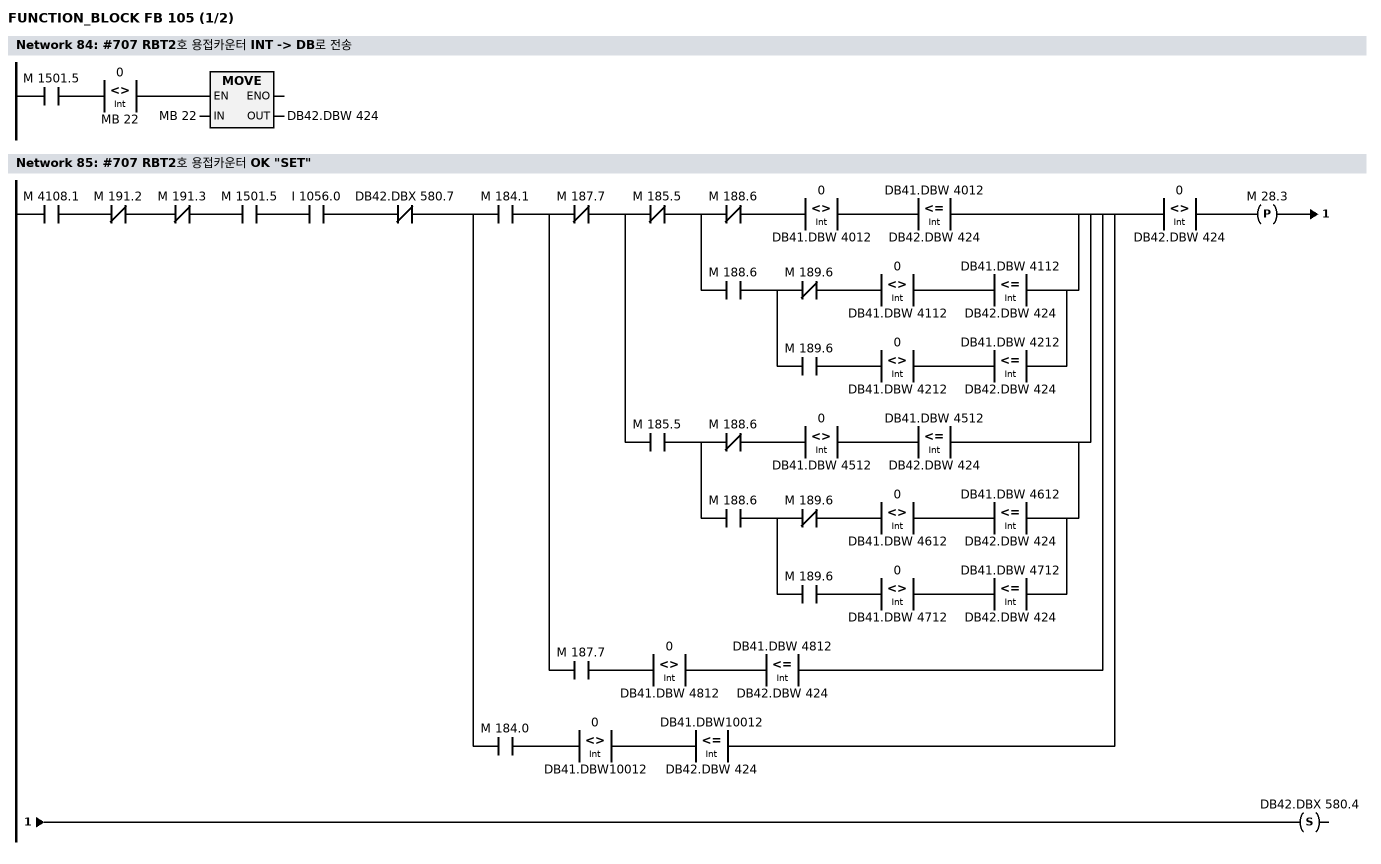

      A     M   1501.5;
      A(    ;
      L     0;
      L     MB    22;
      <>I   ;
      )     ;
      JNB   _093;
      L     MB    22;
      T     DB42.DBW  424;
_093: NOP   0;
NETWORK
TITLE =#707 RBT2호 용접카운터 OK "SET"

      A     M   4108.1;
      AN    M    191.2;
      AN    M    191.3;
      A     M   1501.5;
      A     I   1056.0;
      AN    DB42.DBX  580.7;
      A(    ;
      A     M    184.1;
      A(    ;
      AN    M    187.7;
      A(    ;
      AN    M    185.5;
      A(    ;
      AN    M    188.6;
      A(    ;
      L     0;
      L     DB41.DBW 4012;
      <>I   ;
      )     ;
      A(    ;
      L     DB41.DBW 4012;
      L     DB42.DBW  424;
      <=I   ;
      )     ;
      O     ;
      A     M    188.6;
      A(    ;
      AN    M    189.6;
      A(    ;
      L     0;
      L     DB41.DBW 4112;
      <>I   ;
      )     ;
      A(    ;
      L     DB41.DBW 4112;
      L     DB42.DBW  424;
      <=I   ;
      )     ;
      O     ;
      A     M    189.6;
      A(    ;
      L     0;
      L     DB41.DBW 4212;
      <>I   ;
      )     ;
      A(    ;
      L     DB41.DBW 4212;
      L     DB42.DBW  424;
      <=I   ;
      )     ;
      )     ;
      )     ;
      O     ;
      A     M    185.5;
      A(    ;
      AN    M    188.6;
      A(    ;
      L     0;
      L     DB41.DBW 4512;
      <>I   ;
      )     ;
      A(    ;
      L     DB41.DBW 4512;
      L     DB42.DBW  424;
      <=I   ;
      )     ;
      O     ;
      A     M    188.6;
      A(    ;
      AN    M    189.6;
      A(    ;
      L     0;
      L     DB41.DBW 4612;
      <>I   ;
      )     ;
      A(    ;
      L     DB41.DBW 4612;
      L     DB42.DBW  424;
      <=I   ;
      )     ;
      O     ;
      A     M    189.6;
      A(    ;
      L     0;
      L     DB41.DBW 4712;
      <>I   ;
      )     ;
      A(    ;
      L     DB41.DBW 4712;
      L     DB42.DBW  424;
      <=I   ;
      )     ;
      )     ;
      )     ;
      )     ;
      O     ;
      A     M    187.7;
      A(    ;
      L     0;
      L     DB41.DBW 4812;
      <>I   ;
      )     ;
      A(    ;
      L     DB41.DBW 4812;
      L     DB42.DBW  424;
      <=I   ;
      )     ;
      )     ;
      O     ;
      A     M    184.0;
      A(    ;
      L     0;
      L     DB41.DBW10012;
      <>I   ;
      )     ;
      A(    ;
      L     DB41.DBW10012;
      L     DB42.DBW  424;
      <=I   ;
      )     ;
      )     ;
      A(    ;
      L     0;
      L     DB42.DBW  424;
      <>I   ;
      )     ;
      FP    M     28.3;
      S     DB42.DBX  580.4;
NETWORK
TITLE =#707 RBT2호 용접카운터 NG "SET"
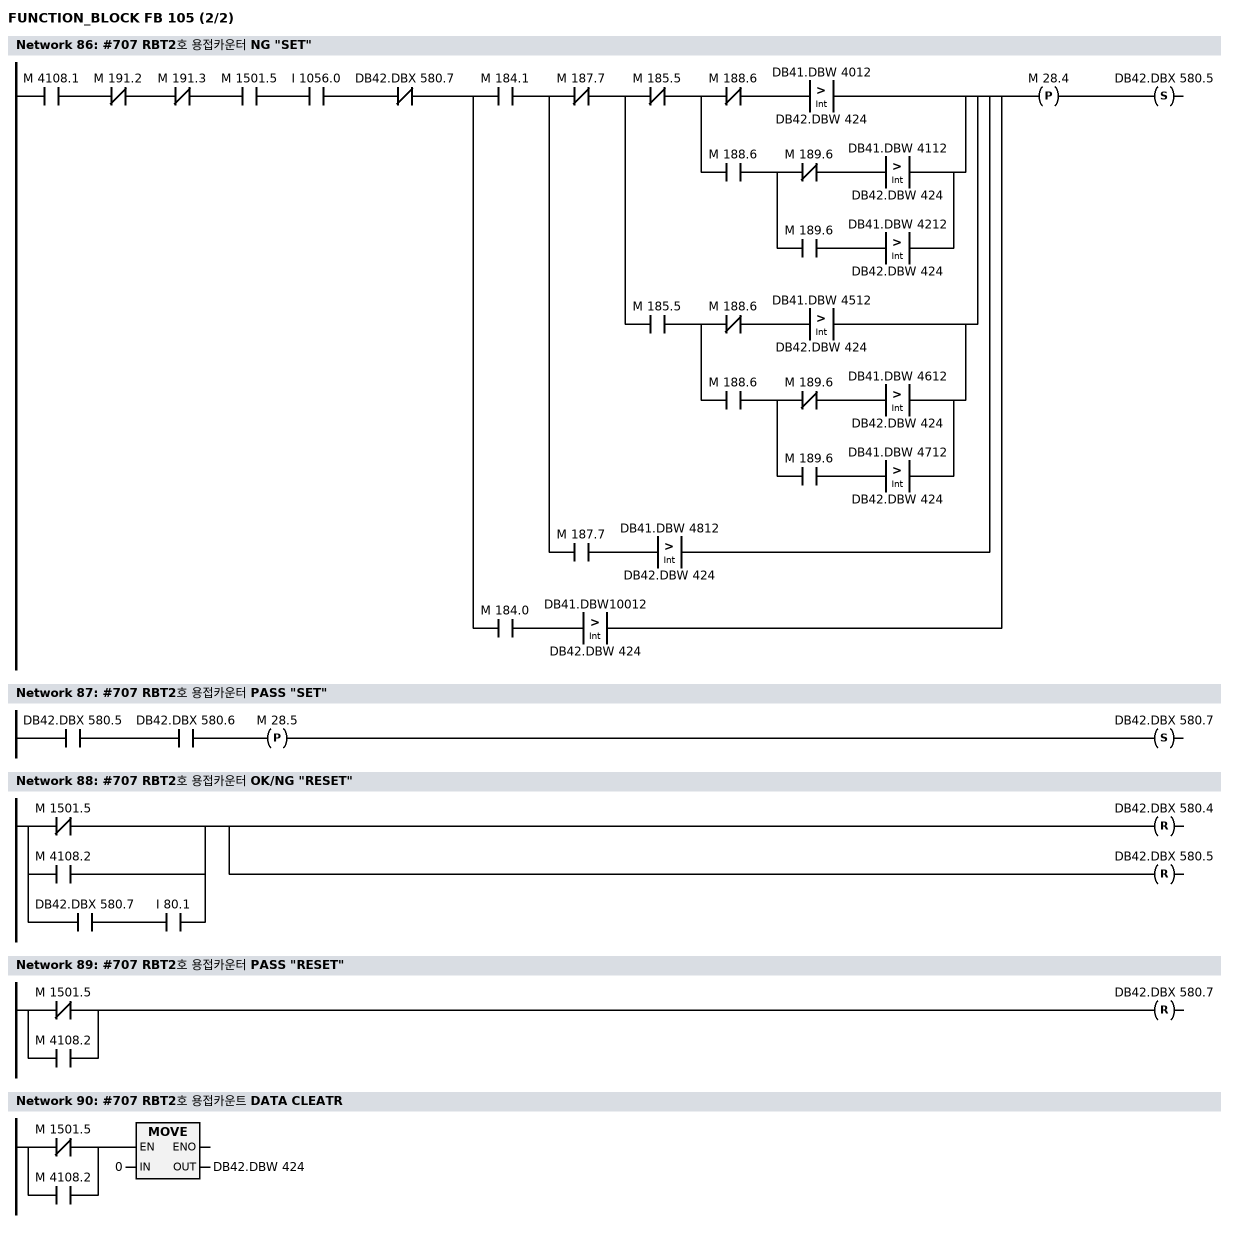

      A     M   4108.1;
      AN    M    191.2;
      AN    M    191.3;
      A     M   1501.5;
      A     I   1056.0;
      AN    DB42.DBX  580.7;
      A(    ;
      A     M    184.1;
      A(    ;
      AN    M    187.7;
      A(    ;
      AN    M    185.5;
      A(    ;
      AN    M    188.6;
      A(    ;
      L     DB41.DBW 4012;
      L     DB42.DBW  424;
      >I    ;
      )     ;
      O     ;
      A     M    188.6;
      A(    ;
      AN    M    189.6;
      A(    ;
      L     DB41.DBW 4112;
      L     DB42.DBW  424;
      >I    ;
      )     ;
      O     ;
      A     M    189.6;
      A(    ;
      L     DB41.DBW 4212;
      L     DB42.DBW  424;
      >I    ;
      )     ;
      )     ;
      )     ;
      O     ;
      A     M    185.5;
      A(    ;
      AN    M    188.6;
      A(    ;
      L     DB41.DBW 4512;
      L     DB42.DBW  424;
      >I    ;
      )     ;
      O     ;
      A     M    188.6;
      A(    ;
      AN    M    189.6;
      A(    ;
      L     DB41.DBW 4612;
      L     DB42.DBW  424;
      >I    ;
      )     ;
      O     ;
      A     M    189.6;
      A(    ;
      L     DB41.DBW 4712;
      L     DB42.DBW  424;
      >I    ;
      )     ;
      )     ;
      )     ;
      )     ;
      O     ;
      A     M    187.7;
      A(    ;
      L     DB41.DBW 4812;
      L     DB42.DBW  424;
      >I    ;
      )     ;
      )     ;
      O     ;
      A     M    184.0;
      A(    ;
      L     DB41.DBW10012;
      L     DB42.DBW  424;
      >I    ;
      )     ;
      )     ;
      FP    M     28.4;
      S     DB42.DBX  580.5;
NETWORK
TITLE =#707 RBT2호 용접카운터 PASS "SET"
//
//
      A     DB42.DBX  580.5;
      A     DB42.DBX  580.6;
      FP    M     28.5;
      S     DB42.DBX  580.7;
NETWORK
TITLE =#707 RBT2호 용접카운터 OK/NG "RESET"

      ON    M   1501.5;
      O     M   4108.2;
      O     ;
      A     DB42.DBX  580.7;
      A     I     80.1;
      R     DB42.DBX  580.4;
      R     DB42.DBX  580.5;
NETWORK
TITLE =#707 RBT2호 용접카운터 PASS "RESET"

      ON    M   1501.5;
      O     M   4108.2;
      R     DB42.DBX  580.7;
NETWORK
TITLE =#707 RBT2호 용접카운트 DATA CLEATR

      A(    ;
      ON    M   1501.5;
      O     M   4108.2;
      )     ;
      JNB   _094;
      L     0;
      T     DB42.DBW  424;
_094: NOP   0;
NETWORK
TITLE =#707 RBT3호 용접카운터 INT -> DB로 전송보조

      AN    OV;
      =     L      2.0;
      A     L      2.0;
      A     I   1068.0;
      =     M     23.0;
      A     L      2.0;
      A     I   1068.1;
      =     M     23.1;
      A     L      2.0;
      A     I   1068.2;
      =     M     23.2;
      A     L      2.0;
      A     I   1068.3;
      =     M     23.3;
      A     L      2.0;
      A     I   1068.4;
      =     M     23.4;
      A     L      2.0;
      AN    M      3.3;
      =     L      2.1;
      A     L      2.1;
      A     I   1068.5;
      =     M     23.5;
      A     L      2.1;
      A     I   1068.6;
      =     M     23.6;
      A     L      2.1;
      A     I   1068.7;
      =     M     23.7;
NETWORK
TITLE =#707 RBT3호 용접카운터 INT -> DB로 전송
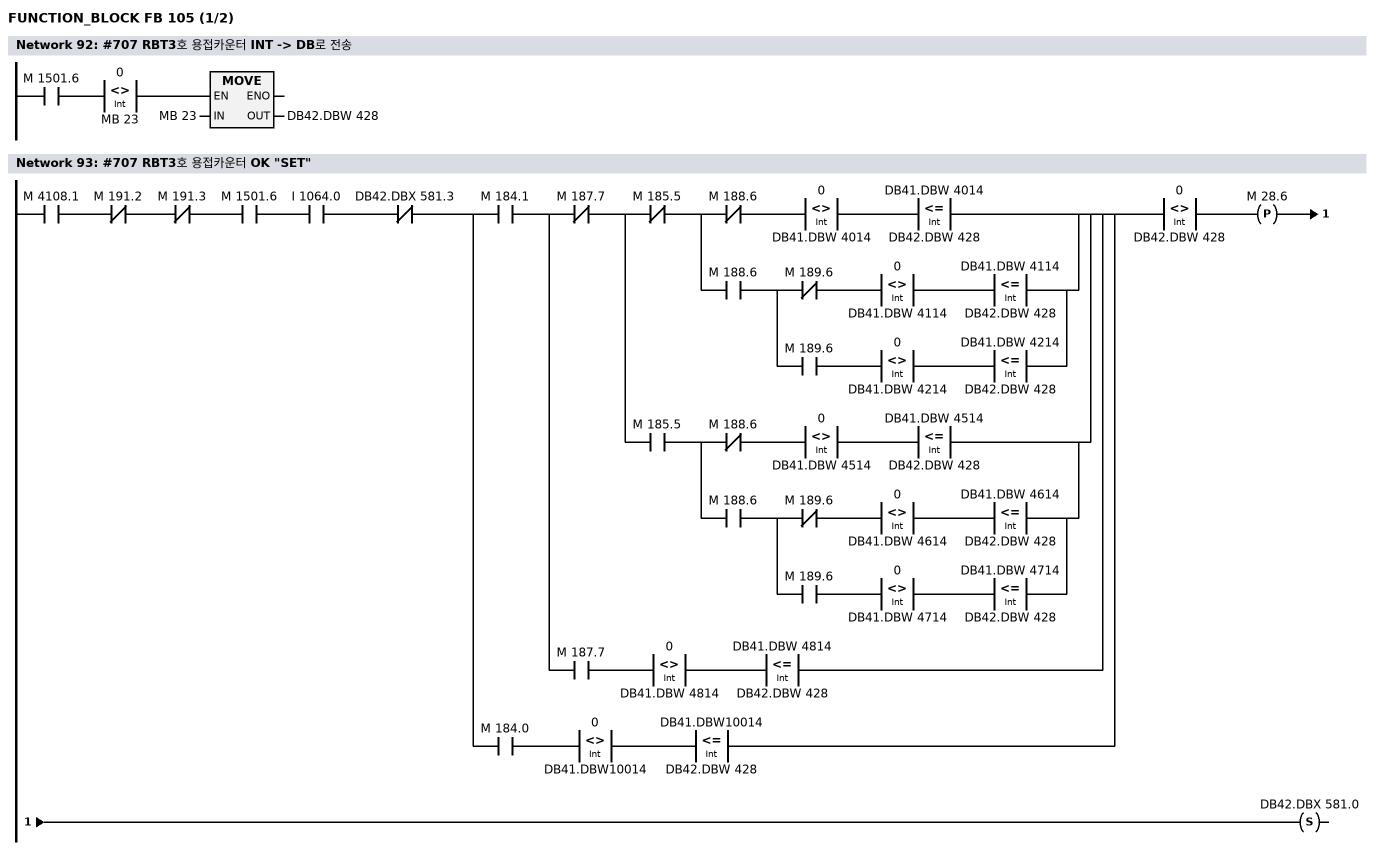

      A     M   1501.6;
      A(    ;
      L     0;
      L     MB    23;
      <>I   ;
      )     ;
      JNB   _095;
      L     MB    23;
      T     DB42.DBW  428;
_095: NOP   0;
NETWORK
TITLE =#707 RBT3호 용접카운터 OK "SET"

      A     M   4108.1;
      AN    M    191.2;
      AN    M    191.3;
      A     M   1501.6;
      A     I   1064.0;
      AN    DB42.DBX  581.3;
      A(    ;
      A     M    184.1;
      A(    ;
      AN    M    187.7;
      A(    ;
      AN    M    185.5;
      A(    ;
      AN    M    188.6;
      A(    ;
      L     0;
      L     DB41.DBW 4014;
      <>I   ;
      )     ;
      A(    ;
      L     DB41.DBW 4014;
      L     DB42.DBW  428;
      <=I   ;
      )     ;
      O     ;
      A     M    188.6;
      A(    ;
      AN    M    189.6;
      A(    ;
      L     0;
      L     DB41.DBW 4114;
      <>I   ;
      )     ;
      A(    ;
      L     DB41.DBW 4114;
      L     DB42.DBW  428;
      <=I   ;
      )     ;
      O     ;
      A     M    189.6;
      A(    ;
      L     0;
      L     DB41.DBW 4214;
      <>I   ;
      )     ;
      A(    ;
      L     DB41.DBW 4214;
      L     DB42.DBW  428;
      <=I   ;
      )     ;
      )     ;
      )     ;
      O     ;
      A     M    185.5;
      A(    ;
      AN    M    188.6;
      A(    ;
      L     0;
      L     DB41.DBW 4514;
      <>I   ;
      )     ;
      A(    ;
      L     DB41.DBW 4514;
      L     DB42.DBW  428;
      <=I   ;
      )     ;
      O     ;
      A     M    188.6;
      A(    ;
      AN    M    189.6;
      A(    ;
      L     0;
      L     DB41.DBW 4614;
      <>I   ;
      )     ;
      A(    ;
      L     DB41.DBW 4614;
      L     DB42.DBW  428;
      <=I   ;
      )     ;
      O     ;
      A     M    189.6;
      A(    ;
      L     0;
      L     DB41.DBW 4714;
      <>I   ;
      )     ;
      A(    ;
      L     DB41.DBW 4714;
      L     DB42.DBW  428;
      <=I   ;
      )     ;
      )     ;
      )     ;
      )     ;
      O     ;
      A     M    187.7;
      A(    ;
      L     0;
      L     DB41.DBW 4814;
      <>I   ;
      )     ;
      A(    ;
      L     DB41.DBW 4814;
      L     DB42.DBW  428;
      <=I   ;
      )     ;
      )     ;
      O     ;
      A     M    184.0;
      A(    ;
      L     0;
      L     DB41.DBW10014;
      <>I   ;
      )     ;
      A(    ;
      L     DB41.DBW10014;
      L     DB42.DBW  428;
      <=I   ;
      )     ;
      )     ;
      A(    ;
      L     0;
      L     DB42.DBW  428;
      <>I   ;
      )     ;
      FP    M     28.6;
      S     DB42.DBX  581.0;
NETWORK
TITLE =#707 RBT3호 용접카운터 NG "SET"
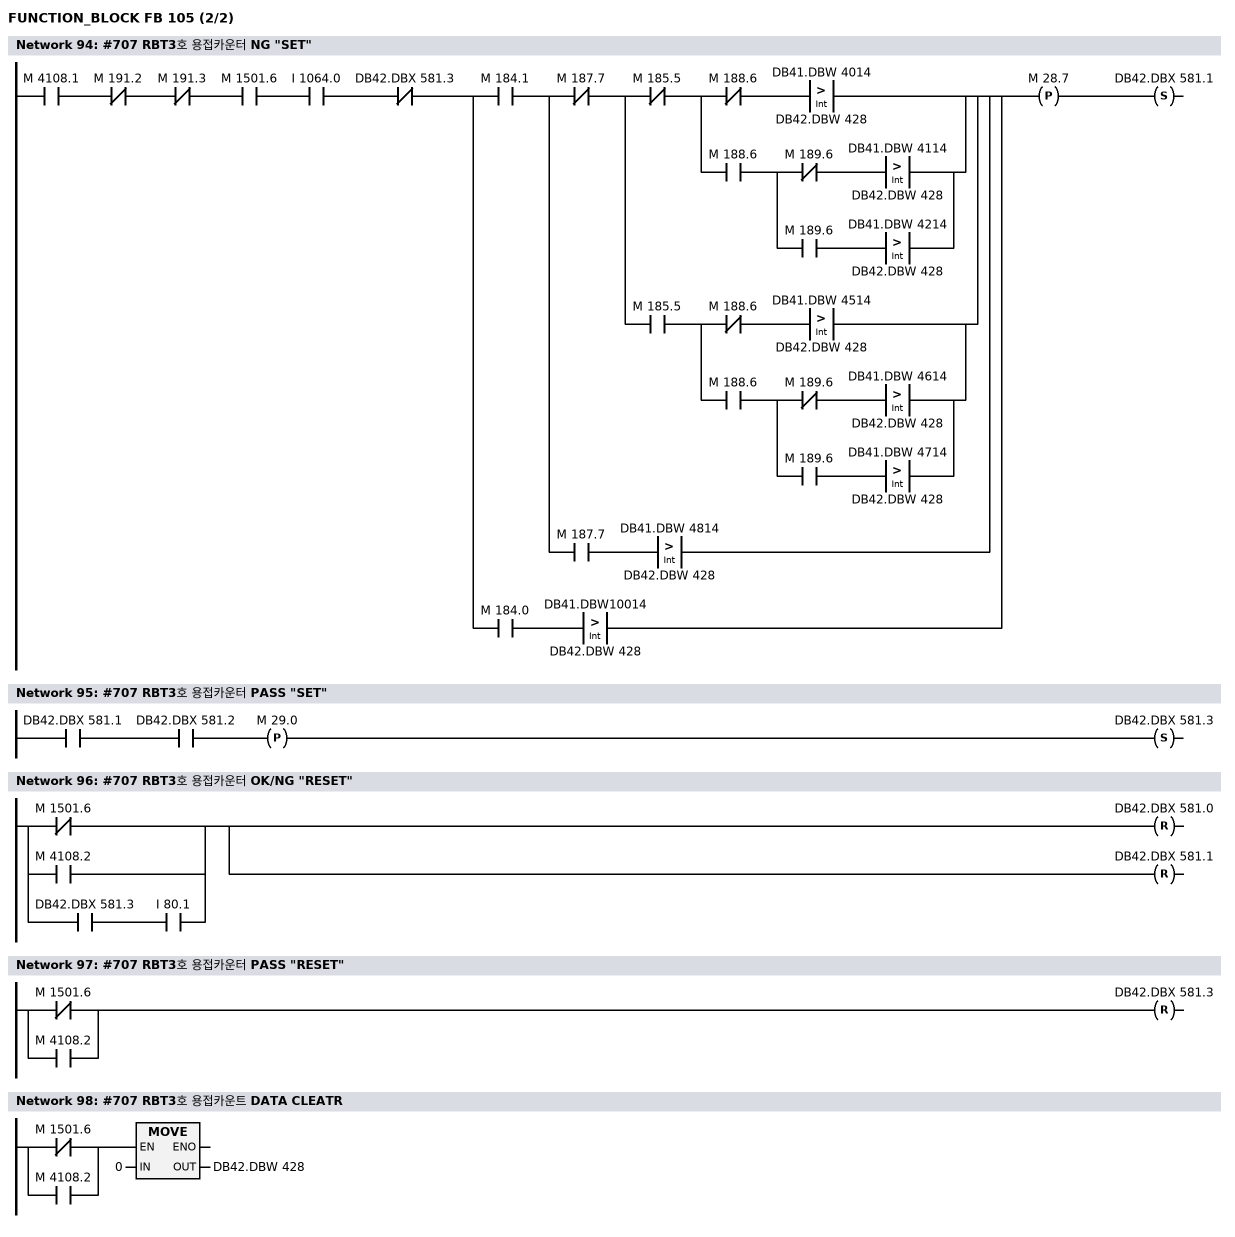

      A     M   4108.1;
      AN    M    191.2;
      AN    M    191.3;
      A     M   1501.6;
      A     I   1064.0;
      AN    DB42.DBX  581.3;
      A(    ;
      A     M    184.1;
      A(    ;
      AN    M    187.7;
      A(    ;
      AN    M    185.5;
      A(    ;
      AN    M    188.6;
      A(    ;
      L     DB41.DBW 4014;
      L     DB42.DBW  428;
      >I    ;
      )     ;
      O     ;
      A     M    188.6;
      A(    ;
      AN    M    189.6;
      A(    ;
      L     DB41.DBW 4114;
      L     DB42.DBW  428;
      >I    ;
      )     ;
      O     ;
      A     M    189.6;
      A(    ;
      L     DB41.DBW 4214;
      L     DB42.DBW  428;
      >I    ;
      )     ;
      )     ;
      )     ;
      O     ;
      A     M    185.5;
      A(    ;
      AN    M    188.6;
      A(    ;
      L     DB41.DBW 4514;
      L     DB42.DBW  428;
      >I    ;
      )     ;
      O     ;
      A     M    188.6;
      A(    ;
      AN    M    189.6;
      A(    ;
      L     DB41.DBW 4614;
      L     DB42.DBW  428;
      >I    ;
      )     ;
      O     ;
      A     M    189.6;
      A(    ;
      L     DB41.DBW 4714;
      L     DB42.DBW  428;
      >I    ;
      )     ;
      )     ;
      )     ;
      )     ;
      O     ;
      A     M    187.7;
      A(    ;
      L     DB41.DBW 4814;
      L     DB42.DBW  428;
      >I    ;
      )     ;
      )     ;
      O     ;
      A     M    184.0;
      A(    ;
      L     DB41.DBW10014;
      L     DB42.DBW  428;
      >I    ;
      )     ;
      )     ;
      FP    M     28.7;
      S     DB42.DBX  581.1;
NETWORK
TITLE =#707 RBT3호 용접카운터 PASS "SET"
//
//
      A     DB42.DBX  581.1;
      A     DB42.DBX  581.2;
      FP    M     29.0;
      S     DB42.DBX  581.3;
NETWORK
TITLE =#707 RBT3호 용접카운터 OK/NG "RESET"

      ON    M   1501.6;
      O     M   4108.2;
      O     ;
      A     DB42.DBX  581.3;
      A     I     80.1;
      R     DB42.DBX  581.0;
      R     DB42.DBX  581.1;
NETWORK
TITLE =#707 RBT3호 용접카운터 PASS "RESET"

      ON    M   1501.6;
      O     M   4108.2;
      R     DB42.DBX  581.3;
NETWORK
TITLE =#707 RBT3호 용접카운트 DATA CLEATR

      A(    ;
      ON    M   1501.6;
      O     M   4108.2;
      )     ;
      JNB   _096;
      L     0;
      T     DB42.DBW  428;
_096: NOP   0;
NETWORK
TITLE =#707 RBT4호 용접카운터 INT -> DB로 전송보조

      AN    OV;
      =     L      2.0;
      A     L      2.0;
      A     I   1076.0;
      =     M     24.0;
      A     L      2.0;
      A     I   1076.1;
      =     M     24.1;
      A     L      2.0;
      A     I   1076.2;
      =     M     24.2;
      A     L      2.0;
      A     I   1076.3;
      =     M     24.3;
      A     L      2.0;
      A     I   1076.4;
      =     M     24.4;
      A     L      2.0;
      AN    M      3.3;
      =     L      2.1;
      A     L      2.1;
      A     I   1076.5;
      =     M     24.5;
      A     L      2.1;
      A     I   1076.6;
      =     M     24.6;
      A     L      2.1;
      A     I   1076.7;
      =     M     24.7;
NETWORK
TITLE =#707 RBT4호 용접카운터 INT -> DB로 전송
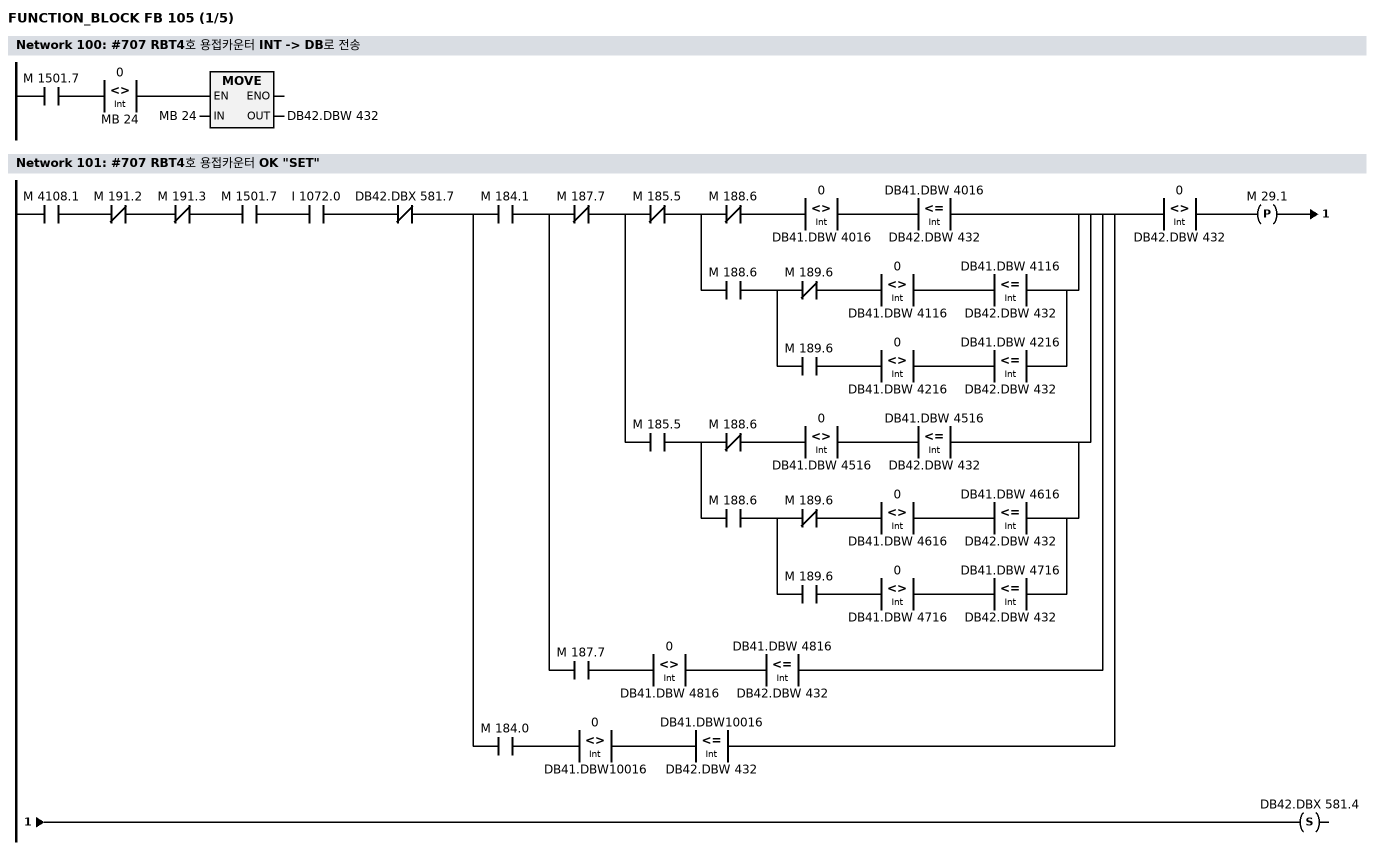

      A     M   1501.7;
      A(    ;
      L     0;
      L     MB    24;
      <>I   ;
      )     ;
      JNB   _097;
      L     MB    24;
      T     DB42.DBW  432;
_097: NOP   0;
NETWORK
TITLE =#707 RBT4호 용접카운터 OK "SET"

      A     M   4108.1;
      AN    M    191.2;
      AN    M    191.3;
      A     M   1501.7;
      A     I   1072.0;
      AN    DB42.DBX  581.7;
      A(    ;
      A     M    184.1;
      A(    ;
      AN    M    187.7;
      A(    ;
      AN    M    185.5;
      A(    ;
      AN    M    188.6;
      A(    ;
      L     0;
      L     DB41.DBW 4016;
      <>I   ;
      )     ;
      A(    ;
      L     DB41.DBW 4016;
      L     DB42.DBW  432;
      <=I   ;
      )     ;
      O     ;
      A     M    188.6;
      A(    ;
      AN    M    189.6;
      A(    ;
      L     0;
      L     DB41.DBW 4116;
      <>I   ;
      )     ;
      A(    ;
      L     DB41.DBW 4116;
      L     DB42.DBW  432;
      <=I   ;
      )     ;
      O     ;
      A     M    189.6;
      A(    ;
      L     0;
      L     DB41.DBW 4216;
      <>I   ;
      )     ;
      A(    ;
      L     DB41.DBW 4216;
      L     DB42.DBW  432;
      <=I   ;
      )     ;
      )     ;
      )     ;
      O     ;
      A     M    185.5;
      A(    ;
      AN    M    188.6;
      A(    ;
      L     0;
      L     DB41.DBW 4516;
      <>I   ;
      )     ;
      A(    ;
      L     DB41.DBW 4516;
      L     DB42.DBW  432;
      <=I   ;
      )     ;
      O     ;
      A     M    188.6;
      A(    ;
      AN    M    189.6;
      A(    ;
      L     0;
      L     DB41.DBW 4616;
      <>I   ;
      )     ;
      A(    ;
      L     DB41.DBW 4616;
      L     DB42.DBW  432;
      <=I   ;
      )     ;
      O     ;
      A     M    189.6;
      A(    ;
      L     0;
      L     DB41.DBW 4716;
      <>I   ;
      )     ;
      A(    ;
      L     DB41.DBW 4716;
      L     DB42.DBW  432;
      <=I   ;
      )     ;
      )     ;
      )     ;
      )     ;
      O     ;
      A     M    187.7;
      A(    ;
      L     0;
      L     DB41.DBW 4816;
      <>I   ;
      )     ;
      A(    ;
      L     DB41.DBW 4816;
      L     DB42.DBW  432;
      <=I   ;
      )     ;
      )     ;
      O     ;
      A     M    184.0;
      A(    ;
      L     0;
      L     DB41.DBW10016;
      <>I   ;
      )     ;
      A(    ;
      L     DB41.DBW10016;
      L     DB42.DBW  432;
      <=I   ;
      )     ;
      )     ;
      A(    ;
      L     0;
      L     DB42.DBW  432;
      <>I   ;
      )     ;
      FP    M     29.1;
      S     DB42.DBX  581.4;
NETWORK
TITLE =#707 RBT4호 용접카운터 NG "SET"
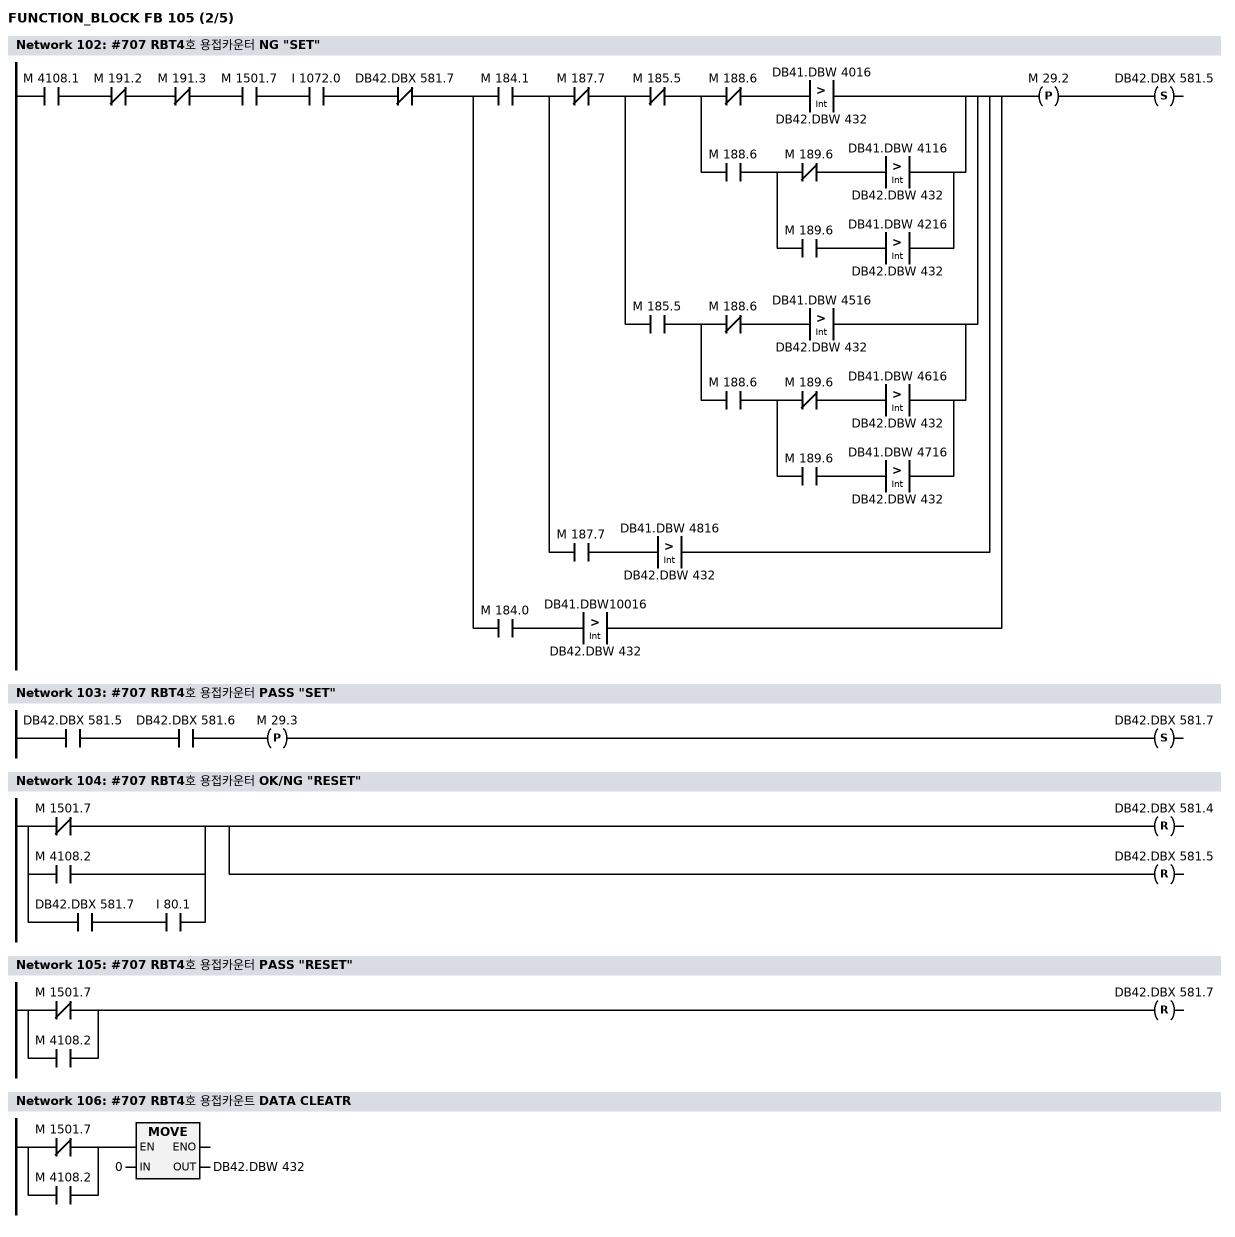

      A     M   4108.1;
      AN    M    191.2;
      AN    M    191.3;
      A     M   1501.7;
      A     I   1072.0;
      AN    DB42.DBX  581.7;
      A(    ;
      A     M    184.1;
      A(    ;
      AN    M    187.7;
      A(    ;
      AN    M    185.5;
      A(    ;
      AN    M    188.6;
      A(    ;
      L     DB41.DBW 4016;
      L     DB42.DBW  432;
      >I    ;
      )     ;
      O     ;
      A     M    188.6;
      A(    ;
      AN    M    189.6;
      A(    ;
      L     DB41.DBW 4116;
      L     DB42.DBW  432;
      >I    ;
      )     ;
      O     ;
      A     M    189.6;
      A(    ;
      L     DB41.DBW 4216;
      L     DB42.DBW  432;
      >I    ;
      )     ;
      )     ;
      )     ;
      O     ;
      A     M    185.5;
      A(    ;
      AN    M    188.6;
      A(    ;
      L     DB41.DBW 4516;
      L     DB42.DBW  432;
      >I    ;
      )     ;
      O     ;
      A     M    188.6;
      A(    ;
      AN    M    189.6;
      A(    ;
      L     DB41.DBW 4616;
      L     DB42.DBW  432;
      >I    ;
      )     ;
      O     ;
      A     M    189.6;
      A(    ;
      L     DB41.DBW 4716;
      L     DB42.DBW  432;
      >I    ;
      )     ;
      )     ;
      )     ;
      )     ;
      O     ;
      A     M    187.7;
      A(    ;
      L     DB41.DBW 4816;
      L     DB42.DBW  432;
      >I    ;
      )     ;
      )     ;
      O     ;
      A     M    184.0;
      A(    ;
      L     DB41.DBW10016;
      L     DB42.DBW  432;
      >I    ;
      )     ;
      )     ;
      FP    M     29.2;
      S     DB42.DBX  581.5;
NETWORK
TITLE =#707 RBT4호 용접카운터 PASS "SET"
//
//
      A     DB42.DBX  581.5;
      A     DB42.DBX  581.6;
      FP    M     29.3;
      S     DB42.DBX  581.7;
NETWORK
TITLE =#707 RBT4호 용접카운터 OK/NG "RESET"

      ON    M   1501.7;
      O     M   4108.2;
      O     ;
      A     DB42.DBX  581.7;
      A     I     80.1;
      R     DB42.DBX  581.4;
      R     DB42.DBX  581.5;
NETWORK
TITLE =#707 RBT4호 용접카운터 PASS "RESET"

      ON    M   1501.7;
      O     M   4108.2;
      R     DB42.DBX  581.7;
NETWORK
TITLE =#707 RBT4호 용접카운트 DATA CLEATR

      A(    ;
      ON    M   1501.7;
      O     M   4108.2;
      )     ;
      JNB   _098;
      L     0;
      T     DB42.DBW  432;
_098: NOP   0;
NETWORK
TITLE =
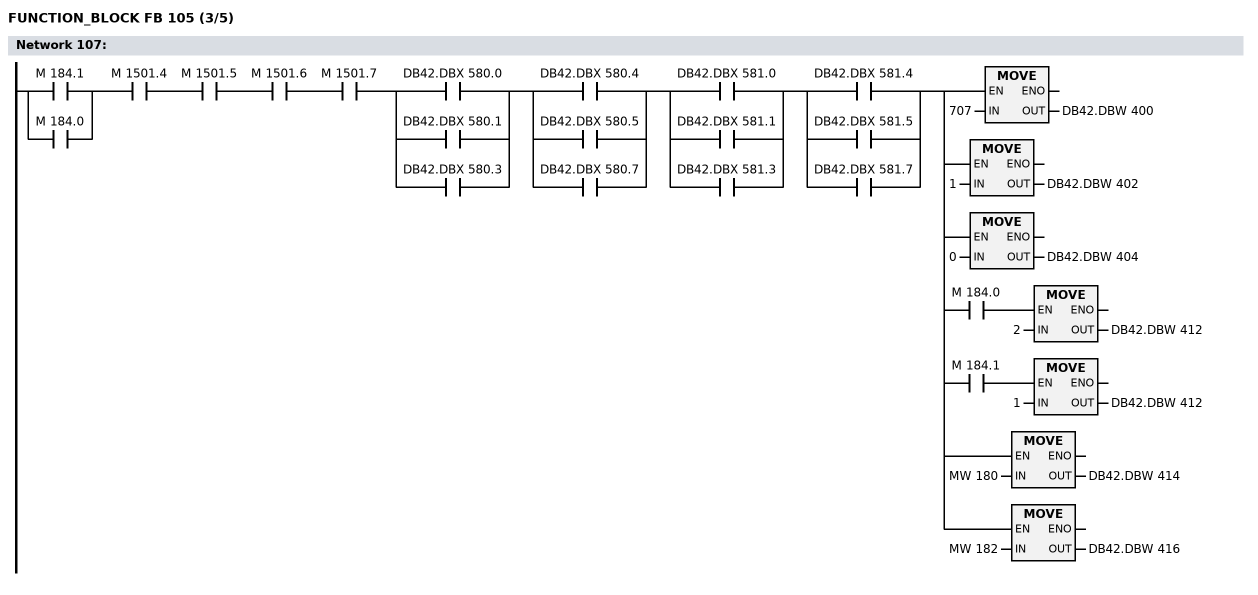

      A(    ;
      O     M    184.1;
      O     M    184.0;
      )     ;
      A     M   1501.4;
      A     M   1501.5;
      A     M   1501.6;
      A     M   1501.7;
      A(    ;
      O     DB42.DBX  580.0;
      O     DB42.DBX  580.1;
      O     DB42.DBX  580.3;
      )     ;
      A(    ;
      O     DB42.DBX  580.4;
      O     DB42.DBX  580.5;
      O     DB42.DBX  580.7;
      )     ;
      A(    ;
      O     DB42.DBX  581.0;
      O     DB42.DBX  581.1;
      O     DB42.DBX  581.3;
      )     ;
      A(    ;
      O     DB42.DBX  581.4;
      O     DB42.DBX  581.5;
      O     DB42.DBX  581.7;
      )     ;
      =     L      2.0;
      A     L      2.0;
      JNB   _099;
      L     707;
      T     DB42.DBW  400;
_099: NOP   0;
      A     L      2.0;
      JNB   _09a;
      L     1;
      T     DB42.DBW  402;
_09a: NOP   0;
      A     L      2.0;
      JNB   _09b;
      L     0;
      T     DB42.DBW  404;
_09b: NOP   0;
      A     L      2.0;
      A     M    184.0;
      JNB   _09c;
      L     2;
      T     DB42.DBW  412;
_09c: NOP   0;
      A     L      2.0;
      A     M    184.1;
      JNB   _09d;
      L     1;
      T     DB42.DBW  412;
_09d: NOP   0;
      A     L      2.0;
      JNB   _09e;
      L     MW   180;
      T     DB42.DBW  414;
_09e: NOP   0;
      A     L      2.0;
      JNB   _09f;
      L     MW   182;
      T     DB42.DBW  416;
_09f: NOP   0;
NETWORK
TITLE =
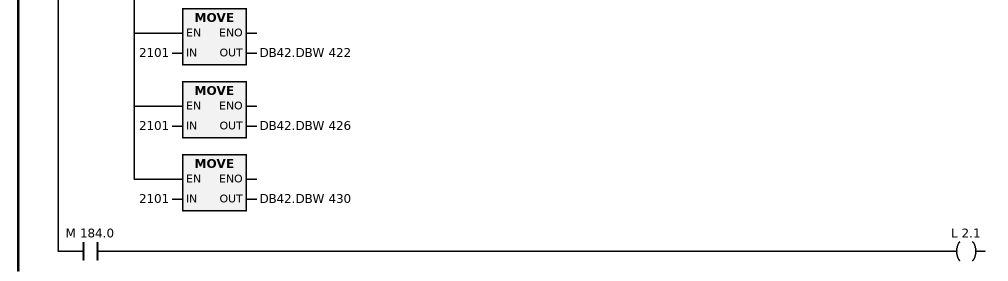

      A(    ;
      O     M    184.1;
      O     M    184.0;
      )     ;
      A     M   1501.4;
      A     M   1501.5;
      A     M   1501.6;
      A     M   1501.7;
      A(    ;
      O     DB42.DBX  580.0;
      O     DB42.DBX  580.1;
      O     DB42.DBX  580.3;
      )     ;
      A(    ;
      O     DB42.DBX  580.4;
      O     DB42.DBX  580.5;
      O     DB42.DBX  580.7;
      )     ;
      A(    ;
      O     DB42.DBX  581.0;
      O     DB42.DBX  581.1;
      O     DB42.DBX  581.3;
      )     ;
      A(    ;
      O     DB42.DBX  581.4;
      O     DB42.DBX  581.5;
      O     DB42.DBX  581.7;
      )     ;
      =     L      2.0;
      A     L      2.0;
      A     M    184.1;
      =     L      2.1;
      A     L      2.1;
      AN    M    187.7;
      =     L      2.2;
      A     L      2.2;
      AN    M    185.5;
      =     L      2.3;
      A     L      2.3;
      AN    M    188.6;
      =     L      2.4;
      A     L      2.4;
      JNB   _0a0;
      L     2011;
      T     DB42.DBW  418;
_0a0: NOP   0;
      A     L      2.4;
      JNB   _0a1;
      L     2011;
      T     DB42.DBW  422;
_0a1: NOP   0;
      A     L      2.4;
      JNB   _0a2;
      L     2011;
      T     DB42.DBW  426;
_0a2: NOP   0;
      A     L      2.4;
      JNB   _0a3;
      L     2011;
      T     DB42.DBW  430;
_0a3: NOP   0;
      A     L      2.3;
      A     M    188.6;
      =     L      2.4;
      A     L      2.4;
      AN    M    189.6;
      =     L      2.5;
      A     L      2.5;
      JNB   _0a4;
      L     2012;
      T     DB42.DBW  418;
_0a4: NOP   0;
      A     L      2.5;
      JNB   _0a5;
      L     2012;
      T     DB42.DBW  422;
_0a5: NOP   0;
      A     L      2.5;
      JNB   _0a6;
      L     2012;
      T     DB42.DBW  426;
_0a6: NOP   0;
      A     L      2.5;
      JNB   _0a7;
      L     2012;
      T     DB42.DBW  430;
_0a7: NOP   0;
      A     L      2.4;
      A     M    189.6;
      =     L      2.5;
      A     L      2.5;
      JNB   _0a8;
      L     2013;
      T     DB42.DBW  418;
_0a8: NOP   0;
      A     L      2.5;
      JNB   _0a9;
      L     2013;
      T     DB42.DBW  422;
_0a9: NOP   0;
      A     L      2.5;
      JNB   _0aa;
      L     2013;
      T     DB42.DBW  426;
_0aa: NOP   0;
      A     L      2.5;
      JNB   _0ab;
      L     2013;
      T     DB42.DBW  430;
_0ab: NOP   0;
      A     L      2.2;
      A     M    185.5;
      =     L      2.3;
      A     L      2.3;
      AN    M    188.6;
      =     L      2.4;
      A     L      2.4;
      JNB   _0ac;
      L     2016;
      T     DB42.DBW  418;
_0ac: NOP   0;
      A     L      2.4;
      JNB   _0ad;
      L     2016;
      T     DB42.DBW  422;
_0ad: NOP   0;
      A     L      2.4;
      JNB   _0ae;
      L     2016;
      T     DB42.DBW  426;
_0ae: NOP   0;
      A     L      2.4;
      JNB   _0af;
      L     2016;
      T     DB42.DBW  430;
_0af: NOP   0;
      A     L      2.3;
      A     M    188.6;
      =     L      2.4;
      A     L      2.4;
      AN    M    189.6;
      =     L      2.5;
      A     L      2.5;
      JNB   _0b0;
      L     2017;
      T     DB42.DBW  418;
_0b0: NOP   0;
      A     L      2.5;
      JNB   _0b1;
      L     2017;
      T     DB42.DBW  422;
_0b1: NOP   0;
      A     L      2.5;
      JNB   _0b2;
      L     2017;
      T     DB42.DBW  426;
_0b2: NOP   0;
      A     L      2.5;
      JNB   _0b3;
      L     2017;
      T     DB42.DBW  430;
_0b3: NOP   0;
      A     L      2.4;
      A     M    189.6;
      =     L      2.5;
      A     L      2.5;
      JNB   _0b4;
      L     2018;
      T     DB42.DBW  418;
_0b4: NOP   0;
      A     L      2.5;
      JNB   _0b5;
      L     2018;
      T     DB42.DBW  422;
_0b5: NOP   0;
      A     L      2.5;
      JNB   _0b6;
      L     2018;
      T     DB42.DBW  426;
_0b6: NOP   0;
      A     L      2.5;
      JNB   _0b7;
      L     2018;
      T     DB42.DBW  430;
_0b7: NOP   0;
      A     L      2.1;
      A     M    187.7;
      =     L      2.2;
      A     L      2.2;
      JNB   _0b8;
      L     2019;
      T     DB42.DBW  418;
_0b8: NOP   0;
      A     L      2.2;
      JNB   _0b9;
      L     2019;
      T     DB42.DBW  422;
_0b9: NOP   0;
      A     L      2.2;
      JNB   _0ba;
      L     2019;
      T     DB42.DBW  426;
_0ba: NOP   0;
      A     L      2.2;
      JNB   _0bb;
      L     2019;
      T     DB42.DBW  430;
_0bb: NOP   0;
      A     L      2.0;
      A     M    184.0;
      =     L      2.1;
      A     L      2.1;
      JNB   _0bc;
      L     2101;
      T     DB42.DBW  418;
_0bc: NOP   0;
      A     L      2.1;
      JNB   _0bd;
      L     2101;
      T     DB42.DBW  422;
_0bd: NOP   0;
      A     L      2.1;
      JNB   _0be;
      L     2101;
      T     DB42.DBW  426;
_0be: NOP   0;
      A     L      2.1;
      JNB   _0bf;
      L     2101;
      T     DB42.DBW  430;
_0bf: NOP   0;
NETWORK
TITLE =
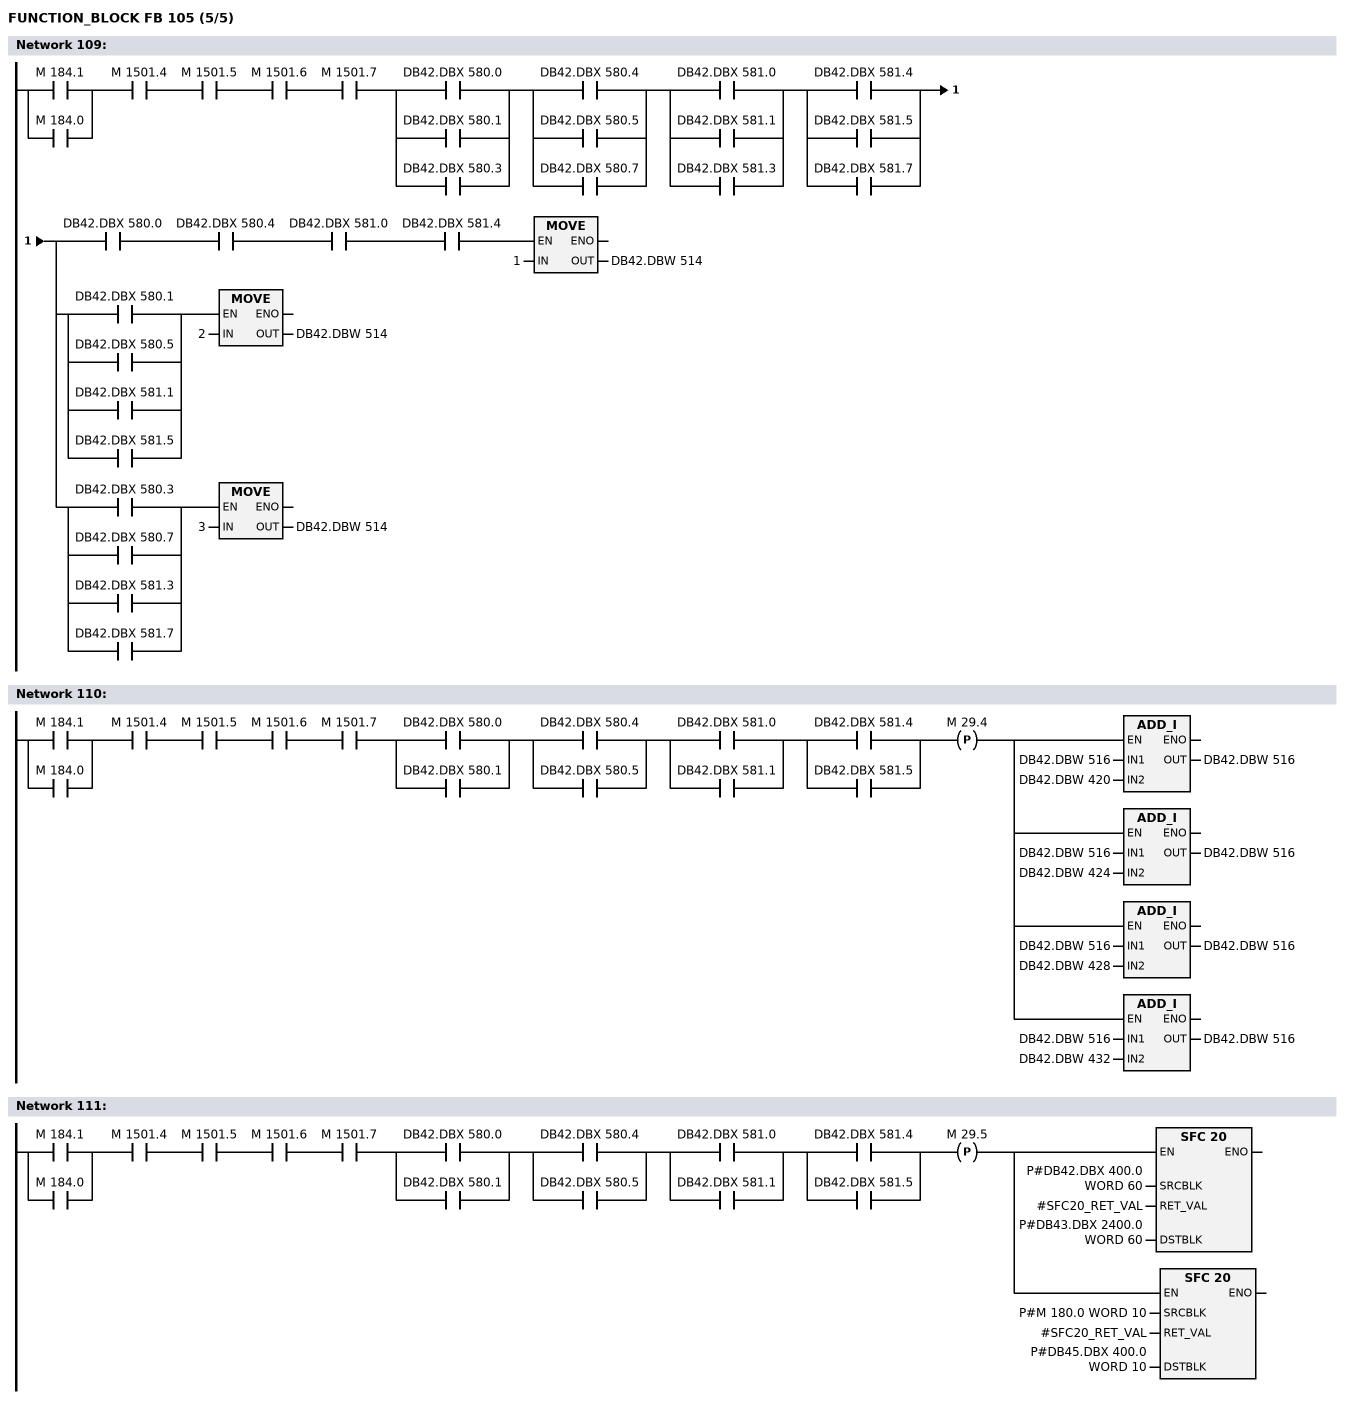

      A(    ;
      O     M    184.1;
      O     M    184.0;
      )     ;
      A     M   1501.4;
      A     M   1501.5;
      A     M   1501.6;
      A     M   1501.7;
      A(    ;
      O     DB42.DBX  580.0;
      O     DB42.DBX  580.1;
      O     DB42.DBX  580.3;
      )     ;
      A(    ;
      O     DB42.DBX  580.4;
      O     DB42.DBX  580.5;
      O     DB42.DBX  580.7;
      )     ;
      A(    ;
      O     DB42.DBX  581.0;
      O     DB42.DBX  581.1;
      O     DB42.DBX  581.3;
      )     ;
      A(    ;
      O     DB42.DBX  581.4;
      O     DB42.DBX  581.5;
      O     DB42.DBX  581.7;
      )     ;
      =     L      2.0;
      A     L      2.0;
      A     DB42.DBX  580.0;
      A     DB42.DBX  580.4;
      A     DB42.DBX  581.0;
      A     DB42.DBX  581.4;
      JNB   _0c0;
      L     1;
      T     DB42.DBW  514;
_0c0: NOP   0;
      A     L      2.0;
      A(    ;
      O     DB42.DBX  580.1;
      O     DB42.DBX  580.5;
      O     DB42.DBX  581.1;
      O     DB42.DBX  581.5;
      )     ;
      JNB   _0c1;
      L     2;
      T     DB42.DBW  514;
_0c1: NOP   0;
      A     L      2.0;
      A(    ;
      O     DB42.DBX  580.3;
      O     DB42.DBX  580.7;
      O     DB42.DBX  581.3;
      O     DB42.DBX  581.7;
      )     ;
      JNB   _0c2;
      L     3;
      T     DB42.DBW  514;
_0c2: NOP   0;
NETWORK
TITLE =

      A(    ;
      O     M    184.1;
      O     M    184.0;
      )     ;
      A     M   1501.4;
      A     M   1501.5;
      A     M   1501.6;
      A     M   1501.7;
      A(    ;
      O     DB42.DBX  580.0;
      O     DB42.DBX  580.1;
      )     ;
      A(    ;
      O     DB42.DBX  580.4;
      O     DB42.DBX  580.5;
      )     ;
      A(    ;
      O     DB42.DBX  581.0;
      O     DB42.DBX  581.1;
      )     ;
      A(    ;
      O     DB42.DBX  581.4;
      O     DB42.DBX  581.5;
      )     ;
      FP    M     29.4;
      =     L      2.0;
      A     L      2.0;
      JNB   _0c3;
      L     DB42.DBW  516;
      L     DB42.DBW  420;
      +I    ;
      T     DB42.DBW  516;
_0c3: NOP   0;
      A     L      2.0;
      JNB   _0c4;
      L     DB42.DBW  516;
      L     DB42.DBW  424;
      +I    ;
      T     DB42.DBW  516;
_0c4: NOP   0;
      A     L      2.0;
      JNB   _0c5;
      L     DB42.DBW  516;
      L     DB42.DBW  428;
      +I    ;
      T     DB42.DBW  516;
_0c5: NOP   0;
      A     L      2.0;
      JNB   _0c6;
      L     DB42.DBW  516;
      L     DB42.DBW  432;
      +I    ;
      T     DB42.DBW  516;
_0c6: NOP   0;
NETWORK
TITLE =

      A(    ;
      O     M    184.1;
      O     M    184.0;
      )     ;
      A     M   1501.4;
      A     M   1501.5;
      A     M   1501.6;
      A     M   1501.7;
      A(    ;
      O     DB42.DBX  580.0;
      O     DB42.DBX  580.1;
      )     ;
      A(    ;
      O     DB42.DBX  580.4;
      O     DB42.DBX  580.5;
      )     ;
      A(    ;
      O     DB42.DBX  581.0;
      O     DB42.DBX  581.1;
      )     ;
      A(    ;
      O     DB42.DBX  581.4;
      O     DB42.DBX  581.5;
      )     ;
      FP    M     29.5;
      =     L      2.0;
      A     L      2.0;
      JNB   _0c7;
      CALL SFC   20 (
           SRCBLK                   := P#DB42.DBX 400.0 WORD 60,
           RET_VAL                  := #SFC20_RET_VAL,
           DSTBLK                   := P#DB43.DBX 2400.0 WORD 60);
_0c7: NOP   0;
      A     L      2.0;
      JNB   _0c8;
      CALL SFC   20 (
           SRCBLK                   := P#M 180.0 WORD 10,
           RET_VAL                  := #SFC20_RET_VAL,
           DSTBLK                   := P#DB45.DBX 400.0 WORD 10);
_0c8: NOP   0;
NETWORK
TITLE =

      A     M   4108.2;
      FP    M     29.6;
      =     L      2.0;
      A(    ;
      A     L      2.0;
      JNB   _0c9;
      CALL SFC   20 (
           SRCBLK                   := P#DB43.DBX 3360.0 WORD 60,
           RET_VAL                  := #SFC20_RET_VAL,
           DSTBLK                   := P#DB43.DBX 3480.0 WORD 60);
_0c9: A     BR;
      )     ;
      JNB   _0ca;
      CALL SFC   20 (
           SRCBLK                   := P#DB43.DBX 3240.0 WORD 60,
           RET_VAL                  := #SFC20_RET_VAL,
           DSTBLK                   := P#DB43.DBX 3360.0 WORD 60);
_0ca: NOP   0;
      A(    ;
      A     L      2.0;
      JNB   _0cb;
      CALL SFC   20 (
           SRCBLK                   := P#DB43.DBX 3120.0 WORD 60,
           RET_VAL                  := #SFC20_RET_VAL,
           DSTBLK                   := P#DB43.DBX 3240.0 WORD 60);
_0cb: A     BR;
      )     ;
      JNB   _0cc;
      CALL SFC   20 (
           SRCBLK                   := P#DB43.DBX 3000.0 WORD 60,
           RET_VAL                  := #SFC20_RET_VAL,
           DSTBLK                   := P#DB43.DBX 3120.0 WORD 60);
_0cc: NOP   0;
      A(    ;
      A     L      2.0;
      JNB   _0cd;
      CALL SFC   20 (
           SRCBLK                   := P#DB43.DBX 2880.0 WORD 60,
           RET_VAL                  := #SFC20_RET_VAL,
           DSTBLK                   := P#DB43.DBX 3000.0 WORD 60);
_0cd: A     BR;
      )     ;
      JNB   _0ce;
      CALL SFC   20 (
           SRCBLK                   := P#DB43.DBX 2760.0 WORD 60,
           RET_VAL                  := #SFC20_RET_VAL,
           DSTBLK                   := P#DB43.DBX 2880.0 WORD 60);
_0ce: NOP   0;
      A(    ;
      A     L      2.0;
      JNB   _0cf;
      CALL SFC   20 (
           SRCBLK                   := P#DB43.DBX 2640.0 WORD 60,
           RET_VAL                  := #SFC20_RET_VAL,
           DSTBLK                   := P#DB43.DBX 2760.0 WORD 60);
_0cf: A     BR;
      )     ;
      JNB   _0d0;
      CALL SFC   20 (
           SRCBLK                   := P#DB43.DBX 2520.0 WORD 60,
           RET_VAL                  := #SFC20_RET_VAL,
           DSTBLK                   := P#DB43.DBX 2640.0 WORD 60);
_0d0: NOP   0;
      A     L      2.0;
      JNB   _0d1;
      CALL SFC   20 (
           SRCBLK                   := P#DB43.DBX 2400.0 WORD 60,
           RET_VAL                  := #SFC20_RET_VAL,
           DSTBLK                   := P#DB43.DBX 2520.0 WORD 60);
_0d1: NOP   0;
      A     L      2.0;
      JNB   _0d2;
      CALL SFC   21 (
           IN0                      := P#M 40.0 WORD 1,
           RET_VAL                  := #SFC20_RET_VAL,
           OUT1                     := P#DB43.DBX 2400.0 WORD 60);
_0d2: NOP   0;
      A(    ;
      A     L      2.0;
      JNB   _0d3;
      CALL SFC   20 (
           SRCBLK                   := P#DB45.DBX 560.0 WORD 10,
           RET_VAL                  := #SFC20_RET_VAL,
           DSTBLK                   := P#DB45.DBX 580.0 WORD 10);
_0d3: A     BR;
      )     ;
      JNB   _0d4;
      CALL SFC   20 (
           SRCBLK                   := P#DB45.DBX 540.0 WORD 10,
           RET_VAL                  := #SFC20_RET_VAL,
           DSTBLK                   := P#DB45.DBX 560.0 WORD 10);
_0d4: NOP   0;
      A(    ;
      A     L      2.0;
      JNB   _0d5;
      CALL SFC   20 (
           SRCBLK                   := P#DB45.DBX 520.0 WORD 10,
           RET_VAL                  := #SFC20_RET_VAL,
           DSTBLK                   := P#DB45.DBX 540.0 WORD 10);
_0d5: A     BR;
      )     ;
      JNB   _0d6;
      CALL SFC   20 (
           SRCBLK                   := P#DB45.DBX 500.0 WORD 10,
           RET_VAL                  := #SFC20_RET_VAL,
           DSTBLK                   := P#DB45.DBX 520.0 WORD 10);
_0d6: NOP   0;
      A(    ;
      A     L      2.0;
      JNB   _0d7;
      CALL SFC   20 (
           SRCBLK                   := P#DB45.DBX 480.0 WORD 10,
           RET_VAL                  := #SFC20_RET_VAL,
           DSTBLK                   := P#DB45.DBX 500.0 WORD 10);
_0d7: A     BR;
      )     ;
      JNB   _0d8;
      CALL SFC   20 (
           SRCBLK                   := P#DB45.DBX 460.0 WORD 10,
           RET_VAL                  := #SFC20_RET_VAL,
           DSTBLK                   := P#DB45.DBX 480.0 WORD 10);
_0d8: NOP   0;
      A(    ;
      A     L      2.0;
      JNB   _0d9;
      CALL SFC   20 (
           SRCBLK                   := P#DB45.DBX 440.0 WORD 10,
           RET_VAL                  := #SFC20_RET_VAL,
           DSTBLK                   := P#DB45.DBX 460.0 WORD 10);
_0d9: A     BR;
      )     ;
      JNB   _0da;
      CALL SFC   20 (
           SRCBLK                   := P#DB45.DBX 420.0 WORD 10,
           RET_VAL                  := #SFC20_RET_VAL,
           DSTBLK                   := P#DB45.DBX 440.0 WORD 10);
_0da: NOP   0;
      A     L      2.0;
      JNB   _0db;
      CALL SFC   20 (
           SRCBLK                   := P#DB45.DBX 400.0 WORD 10,
           RET_VAL                  := #SFC20_RET_VAL,
           DSTBLK                   := P#DB45.DBX 420.0 WORD 10);
_0db: NOP   0;
      A     L      2.0;
      JNB   _0dc;
      CALL SFC   21 (
           IN0                      := P#M 40.0 WORD 1,
           RET_VAL                  := #SFC20_RET_VAL,
           OUT1                     := P#DB45.DBX 400.0 WORD 10);
_0dc: NOP   0;
NETWORK
TITLE =
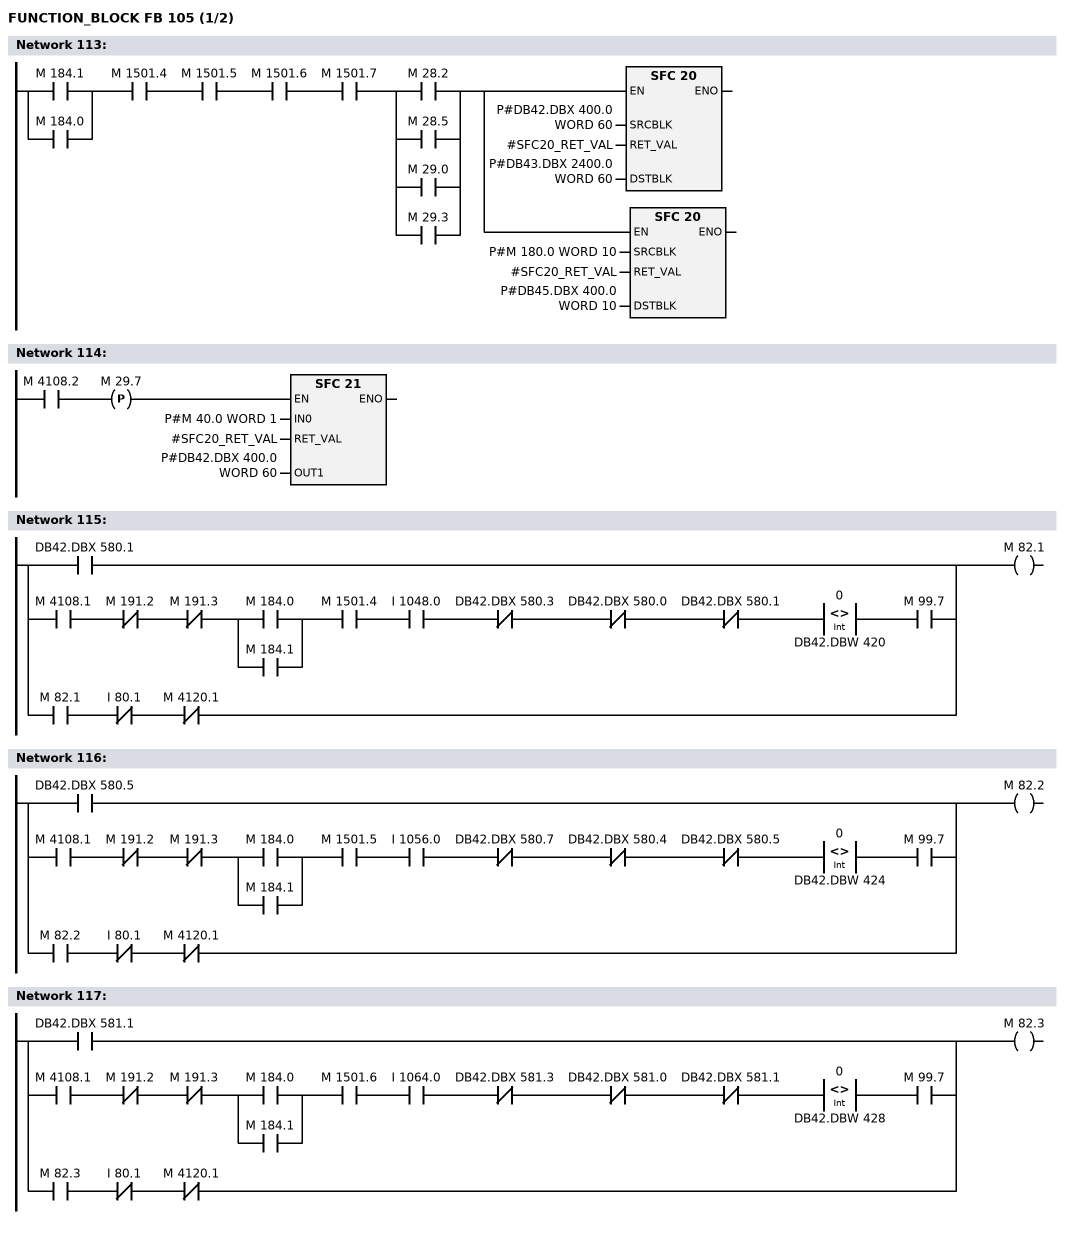

      A(    ;
      O     M    184.1;
      O     M    184.0;
      )     ;
      A     M   1501.4;
      A     M   1501.5;
      A     M   1501.6;
      A     M   1501.7;
      A(    ;
      O     M     28.2;
      O     M     28.5;
      O     M     29.0;
      O     M     29.3;
      )     ;
      =     L      2.0;
      A     L      2.0;
      JNB   _0dd;
      CALL SFC   20 (
           SRCBLK                   := P#DB42.DBX 400.0 WORD 60,
           RET_VAL                  := #SFC20_RET_VAL,
           DSTBLK                   := P#DB43.DBX 2400.0 WORD 60);
_0dd: NOP   0;
      A     L      2.0;
      JNB   _0de;
      CALL SFC   20 (
           SRCBLK                   := P#M 180.0 WORD 10,
           RET_VAL                  := #SFC20_RET_VAL,
           DSTBLK                   := P#DB45.DBX 400.0 WORD 10);
_0de: NOP   0;
NETWORK
TITLE =

      A     M   4108.2;
      FP    M     29.7;
      JNB   _0df;
      CALL SFC   21 (
           IN0                      := P#M 40.0 WORD 1,
           RET_VAL                  := #SFC20_RET_VAL,
           OUT1                     := P#DB42.DBX 400.0 WORD 60);
_0df: NOP   0;
NETWORK
TITLE =

      O     DB42.DBX  580.1;
      O     ;
      A     M   4108.1;
      AN    M    191.2;
      AN    M    191.3;
      A(    ;
      O     M    184.0;
      O     M    184.1;
      )     ;
      A     M   1501.4;
      A     I   1048.0;
      AN    DB42.DBX  580.3;
      AN    DB42.DBX  580.0;
      AN    DB42.DBX  580.1;
      A(    ;
      L     0;
      L     DB42.DBW  420;
      <>I   ;
      )     ;
      A     M     99.7;
      O     ;
      A     M     82.1;
      AN    I     80.1;
      AN    M   4120.1;
      =     M     82.1;
NETWORK
TITLE =

      O     DB42.DBX  580.5;
      O     ;
      A     M   4108.1;
      AN    M    191.2;
      AN    M    191.3;
      A(    ;
      O     M    184.0;
      O     M    184.1;
      )     ;
      A     M   1501.5;
      A     I   1056.0;
      AN    DB42.DBX  580.7;
      AN    DB42.DBX  580.4;
      AN    DB42.DBX  580.5;
      A(    ;
      L     0;
      L     DB42.DBW  424;
      <>I   ;
      )     ;
      A     M     99.7;
      O     ;
      A     M     82.2;
      AN    I     80.1;
      AN    M   4120.1;
      =     M     82.2;
NETWORK
TITLE =

      O     DB42.DBX  581.1;
      O     ;
      A     M   4108.1;
      AN    M    191.2;
      AN    M    191.3;
      A(    ;
      O     M    184.0;
      O     M    184.1;
      )     ;
      A     M   1501.6;
      A     I   1064.0;
      AN    DB42.DBX  581.3;
      AN    DB42.DBX  581.0;
      AN    DB42.DBX  581.1;
      A(    ;
      L     0;
      L     DB42.DBW  428;
      <>I   ;
      )     ;
      A     M     99.7;
      O     ;
      A     M     82.3;
      AN    I     80.1;
      AN    M   4120.1;
      =     M     82.3;
NETWORK
TITLE =
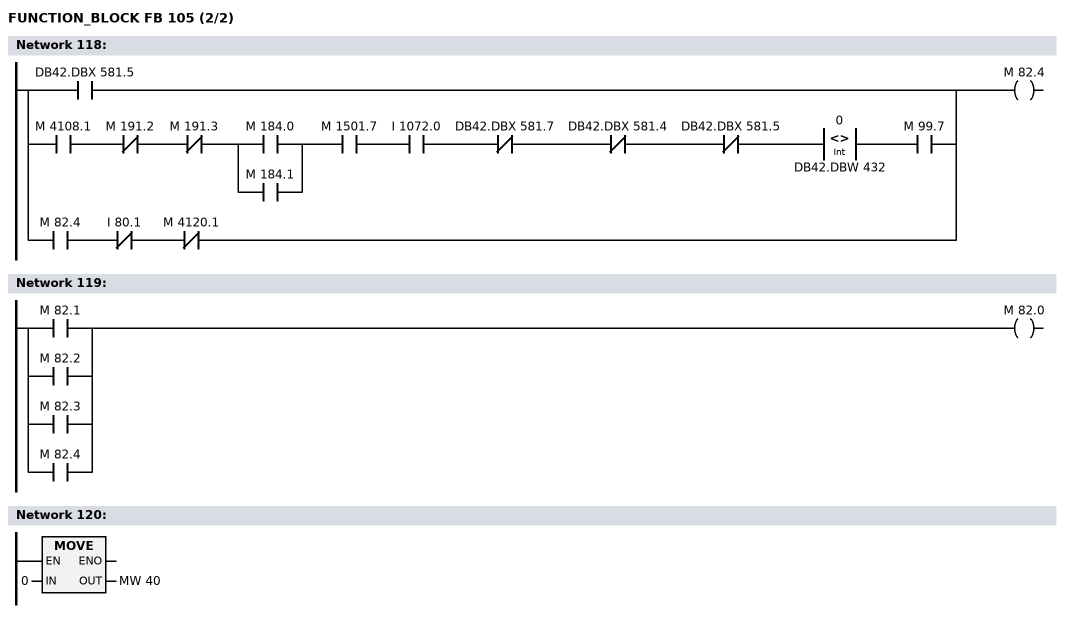

      O     DB42.DBX  581.5;
      O     ;
      A     M   4108.1;
      AN    M    191.2;
      AN    M    191.3;
      A(    ;
      O     M    184.0;
      O     M    184.1;
      )     ;
      A     M   1501.7;
      A     I   1072.0;
      AN    DB42.DBX  581.7;
      AN    DB42.DBX  581.4;
      AN    DB42.DBX  581.5;
      A(    ;
      L     0;
      L     DB42.DBW  432;
      <>I   ;
      )     ;
      A     M     99.7;
      O     ;
      A     M     82.4;
      AN    I     80.1;
      AN    M   4120.1;
      =     M     82.4;
NETWORK
TITLE =

      O     M     82.1;
      O     M     82.2;
      O     M     82.3;
      O     M     82.4;
      =     M     82.0;
NETWORK
TITLE =

      L     0;
      T     MW    40;
      NOP   0;
END_FUNCTION_BLOCK

DATA_BLOCK DB 105
TITLE =
VERSION : 0.0

 FB 105
BEGIN
   S705_RBT1_WELD_OK_PLS := FALSE;
   S705_RBT1_WELD_NG_PLS := FALSE;
   S705_RBT1_WELD_PASS_PLS := FALSE;
   S705_CHECK_SUM_PLS := FALSE;
   S705_WELD_DATA_MOV_BUFF := FALSE;
   MW_0_BUFF[0] := W#16#0;
   MW_0_BUFF[1] := W#16#0;
   MW_0_BUFF[2] := W#16#0;
   MW_0_BUFF[3] := W#16#0;
   MW_0_BUFF[4] := W#16#0;
   MW_0_BUFF[5] := W#16#0;
   MW_0_BUFF[6] := W#16#0;
   MW_0_BUFF[7] := W#16#0;
   MW_0_BUFF[8] := W#16#0;
   MW_0_BUFF[9] := W#16#0;
   MW_0_BUFF[10] := W#16#0;
   MW_0_BUFF[11] := W#16#0;
   MW_0_BUFF[12] := W#16#0;
   MW_0_BUFF[13] := W#16#0;
   MW_0_BUFF[14] := W#16#0;
   MW_0_BUFF[15] := W#16#0;
   MW_0_BUFF[16] := W#16#0;
   MW_0_BUFF[17] := W#16#0;
   MW_0_BUFF[18] := W#16#0;
   MW_0_BUFF[19] := W#16#0;
   MW_0_BUFF[20] := W#16#0;
   MW_0_BUFF[21] := W#16#0;
   MW_0_BUFF[22] := W#16#0;
   MW_0_BUFF[23] := W#16#0;
   MW_0_BUFF[24] := W#16#0;
   MW_0_BUFF[25] := W#16#0;
   MW_0_BUFF[26] := W#16#0;
   MW_0_BUFF[27] := W#16#0;
   MW_0_BUFF[28] := W#16#0;
   MW_0_BUFF[29] := W#16#0;
   MW_0_BUFF[30] := W#16#0;
   MW_0_BUFF[31] := W#16#0;
   MW_0_BUFF[32] := W#16#0;
   MW_0_BUFF[33] := W#16#0;
   MW_0_BUFF[34] := W#16#0;
   MW_0_BUFF[35] := W#16#0;
   MW_0_BUFF[36] := W#16#0;
   MW_0_BUFF[37] := W#16#0;
   MW_0_BUFF[38] := W#16#0;
   MW_0_BUFF[39] := W#16#0;
   MW_0_BUFF[40] := W#16#0;
   MW_0_BUFF[41] := W#16#0;
   MW_0_BUFF[42] := W#16#0;
   MW_0_BUFF[43] := W#16#0;
   MW_0_BUFF[44] := W#16#0;
   MW_0_BUFF[45] := W#16#0;
   MW_0_BUFF[46] := W#16#0;
   MW_0_BUFF[47] := W#16#0;
   MW_0_BUFF[48] := W#16#0;
   MW_0_BUFF[49] := W#16#0;
   MW_0_BUFF[50] := W#16#0;
   MW_0_BUFF[51] := W#16#0;
   MW_0_BUFF[52] := W#16#0;
   MW_0_BUFF[53] := W#16#0;
   MW_0_BUFF[54] := W#16#0;
   MW_0_BUFF[55] := W#16#0;
   MW_0_BUFF[56] := W#16#0;
   MW_0_BUFF[57] := W#16#0;
   MW_0_BUFF[58] := W#16#0;
   MW_0_BUFF[59] := W#16#0;
   S706_RBT1_WELD_OK_PLS := FALSE;
   S706_RBT1_WELD_NG_PLS := FALSE;
   S706_RBT1_WELD_PASS_PLS := FALSE;
   S706_RBT2_WELD_OK_PLS := FALSE;
   S706_RBT2_WELD_NG_PLS := FALSE;
   S706_RBT2_WELD_PASS_PLS := FALSE;
   S706_RBT3_WELD_OK_PLS := FALSE;
   S706_RBT3_WELD_NG_PLS := FALSE;
   S706_RBT3_WELD_PASS_PLS := FALSE;
   S706_CHECK_SUM_PLS := FALSE;
   S706_WELD_DATA_MOV_BUFF := FALSE;
   S711_RBT1_WELD_OK_PLS := FALSE;
   S711_RBT1_WELD_NG_PLS := FALSE;
   S711_RBT1_WELD_PASS_PLS := FALSE;
   S711_CHECK_SUM_PLS := FALSE;
   S711_WELD_DATA_MOV_BUFF := FALSE;
   PLS1 := FALSE;
   PLS2 := FALSE;
   PLS3 := FALSE;
   PLS4 := FALSE;
   PLS5 := FALSE;
   PLS6 := FALSE;
END_DATA_BLOCK

FUNCTION_BLOCK FB 108
TITLE =
VERSION : 0.1

BEGIN
NETWORK
TITLE =PROFINET ERROR(1~10)
//
//
      A     M      3.3;
      =     L      0.0;
      A     L      0.0;
      A(    ;
      O     DB327.DBX 1025.3;
      O     ;
      A     M   7000.0;
      AN    I      0.1;
      AN    I     80.1;
      )     ;
      =     L      0.1;
      A     L      0.1;
      A     T    700;
      =     M   7000.0;
      A     L      0.1;
      BLD   102;
      L     S5T#0MS;
      SD    T    700;
      A     L      0.0;
      A(    ;
      O     DB327.DBX 1027.3;
      O     ;
      A     M   7000.1;
      AN    I      0.1;
      AN    I     80.1;
      )     ;
      =     L      0.1;
      A     L      0.1;
      A     T    701;
      =     M   7000.1;
      A     L      0.1;
      BLD   102;
      L     S5T#0MS;
      SD    T    701;
      A     L      0.0;
      A(    ;
      O     DB327.DBX 1029.3;
      O     ;
      A     M   7000.2;
      AN    I      0.1;
      AN    I     80.1;
      )     ;
      =     L      0.1;
      A     L      0.1;
      A     T    702;
      =     M   7000.2;
      A     L      0.1;
      BLD   102;
      L     S5T#0MS;
      SD    T    702;
      A     L      0.0;
      A(    ;
      O     DB327.DBX 1031.3;
      O     ;
      A     M   7000.3;
      AN    I      0.1;
      AN    I     80.1;
      )     ;
      =     L      0.1;
      A     L      0.1;
      A     T    703;
      =     M   7000.3;
      A     L      0.1;
      BLD   102;
      L     S5T#0MS;
      SD    T    703;
      A     L      0.0;
      A(    ;
      O     DB327.DBX 1033.3;
      O     ;
      A     M   7000.4;
      AN    I      0.1;
      AN    I     80.1;
      )     ;
      =     L      0.1;
      A     L      0.1;
      A     T    704;
      =     M   7000.4;
      A     L      0.1;
      BLD   102;
      L     S5T#0MS;
      SD    T    704;
      A     L      0.0;
      A(    ;
      O     DB327.DBX 1035.3;
      O     ;
      A     M   7000.5;
      AN    I      0.1;
      AN    I     80.1;
      )     ;
      =     L      0.1;
      A     L      0.1;
      A     T    705;
      =     M   7000.5;
      A     L      0.1;
      BLD   102;
      L     S5T#0MS;
      SD    T    705;
      A     L      0.0;
      A(    ;
      O     DB327.DBX 1037.3;
      O     ;
      A     M   7000.6;
      AN    I      0.1;
      AN    I     80.1;
      )     ;
      =     L      0.1;
      A     L      0.1;
      A     T    706;
      =     M   7000.6;
      A     L      0.1;
      BLD   102;
      L     S5T#0MS;
      SD    T    706;
      A     L      0.0;
      A(    ;
      O     DB327.DBX 1039.3;
      O     ;
      A     M   7000.7;
      AN    I      0.1;
      AN    I     80.1;
      )     ;
      =     L      0.1;
      A     L      0.1;
      A     T    707;
      =     M   7000.7;
      A     L      0.1;
      BLD   102;
      L     S5T#0MS;
      SD    T    707;
      A     L      0.0;
      A(    ;
      O     DB327.DBX 1041.3;
      O     ;
      A     M   7001.0;
      AN    I      0.1;
      AN    I     80.1;
      )     ;
      =     L      0.1;
      A     L      0.1;
      A     T    708;
      =     M   7001.0;
      A     L      0.1;
      BLD   102;
      L     S5T#0MS;
      SD    T    708;
      A     L      0.0;
      A(    ;
      O     DB327.DBX 1043.3;
      O     ;
      A     M   7001.1;
      AN    I      0.1;
      AN    I     80.1;
      )     ;
      =     L      0.1;
      A     L      0.1;
      A     T    709;
      =     M   7001.1;
      A     L      0.1;
      BLD   102;
      L     S5T#0MS;
      SD    T    709;
NETWORK
TITLE =PROFINET ERROR(11~20)
//
//
      A     M      3.3;
      =     L      0.0;
      A     L      0.0;
      A(    ;
      O     DB327.DBX 1045.3;
      O     ;
      A     M   7001.2;
      AN    I      0.1;
      AN    I     80.1;
      )     ;
      =     L      0.1;
      A     L      0.1;
      A     T    710;
      =     M   7001.2;
      A     L      0.1;
      BLD   102;
      L     S5T#0MS;
      SD    T    710;
      A     L      0.0;
      A(    ;
      O     DB327.DBX 1047.3;
      O     ;
      A     M   7001.3;
      AN    I      0.1;
      AN    I     80.1;
      )     ;
      =     L      0.1;
      A     L      0.1;
      A     T    711;
      =     M   7001.3;
      A     L      0.1;
      BLD   102;
      L     S5T#0MS;
      SD    T    711;
      A     L      0.0;
      A(    ;
      O     DB327.DBX 1049.3;
      O     ;
      A     M   7001.4;
      AN    I      0.1;
      AN    I     80.1;
      )     ;
      =     L      0.1;
      A     L      0.1;
      A     T    712;
      =     M   7001.4;
      A     L      0.1;
      BLD   102;
      L     S5T#0MS;
      SD    T    712;
      A     L      0.0;
      A(    ;
      O     DB327.DBX 1051.3;
      O     ;
      A     M   7001.5;
      AN    I      0.1;
      AN    I     80.1;
      )     ;
      =     L      0.1;
      A     L      0.1;
      A     T    713;
      =     M   7001.5;
      A     L      0.1;
      BLD   102;
      L     S5T#0MS;
      SD    T    713;
      A     L      0.0;
      A(    ;
      O     DB327.DBX 1053.3;
      O     ;
      A     M   7001.6;
      AN    I      0.1;
      AN    I     80.1;
      )     ;
      =     L      0.1;
      A     L      0.1;
      A     T    714;
      =     M   7001.6;
      A     L      0.1;
      BLD   102;
      L     S5T#0MS;
      SD    T    714;
      A     L      0.0;
      A(    ;
      O     DB327.DBX 1055.3;
      O     ;
      A     M   7001.7;
      AN    I      0.1;
      AN    I     80.1;
      )     ;
      =     L      0.1;
      A     L      0.1;
      A     T    715;
      =     M   7001.7;
      A     L      0.1;
      BLD   102;
      L     S5T#0MS;
      SD    T    715;
      A     L      0.0;
      A(    ;
      O     DB327.DBX 1057.3;
      O     ;
      A     M   7002.0;
      AN    I      0.1;
      AN    I     80.1;
      )     ;
      =     L      0.1;
      A     L      0.1;
      A     T    716;
      =     M   7002.0;
      A     L      0.1;
      BLD   102;
      L     S5T#0MS;
      SD    T    716;
      A     L      0.0;
      A(    ;
      O     DB327.DBX 1059.3;
      O     ;
      A     M   7002.1;
      AN    I      0.1;
      AN    I     80.1;
      )     ;
      =     L      0.1;
      A     L      0.1;
      A     T    717;
      =     M   7002.1;
      A     L      0.1;
      BLD   102;
      L     S5T#0MS;
      SD    T    717;
      A     L      0.0;
      A(    ;
      O     DB327.DBX 1061.3;
      O     ;
      A     M   7002.2;
      AN    I      0.1;
      AN    I     80.1;
      )     ;
      =     L      0.1;
      A     L      0.1;
      A     T    718;
      =     M   7002.2;
      A     L      0.1;
      BLD   102;
      L     S5T#0MS;
      SD    T    718;
      A     L      0.0;
      A(    ;
      O     DB327.DBX 1063.3;
      O     ;
      A     M   7002.3;
      AN    I      0.1;
      AN    I     80.1;
      )     ;
      =     L      0.1;
      A     L      0.1;
      A     T    719;
      =     M   7002.3;
      A     L      0.1;
      BLD   102;
      L     S5T#0MS;
      SD    T    719;
NETWORK
TITLE =PROFINET ERROR(21~30)
//
//
      A     M      3.3;
      =     L      0.0;
      A     L      0.0;
      A(    ;
      O     DB327.DBX 1065.3;
      O     ;
      A     M   7002.4;
      AN    I      0.1;
      AN    I     80.1;
      )     ;
      =     L      0.1;
      A     L      0.1;
      A     T    720;
      =     M   7002.4;
      A     L      0.1;
      BLD   102;
      L     S5T#0MS;
      SD    T    720;
      A     L      0.0;
      A(    ;
      O     DB327.DBX 1067.3;
      O     ;
      A     M   7002.5;
      AN    I      0.1;
      AN    I     80.1;
      )     ;
      =     L      0.1;
      A     L      0.1;
      A     T    721;
      =     M   7002.5;
      A     L      0.1;
      BLD   102;
      L     S5T#0MS;
      SD    T    721;
      A     L      0.0;
      A(    ;
      O     DB327.DBX 1069.3;
      O     ;
      A     M   7002.6;
      AN    I      0.1;
      AN    I     80.1;
      )     ;
      =     L      0.1;
      A     L      0.1;
      A     T    722;
      =     M   7002.6;
      A     L      0.1;
      BLD   102;
      L     S5T#0MS;
      SD    T    722;
      A     L      0.0;
      A(    ;
      O     DB327.DBX 1071.3;
      O     ;
      A     M   7002.7;
      AN    I      0.1;
      AN    I     80.1;
      )     ;
      =     L      0.1;
      A     L      0.1;
      A     T    723;
      AN    M      3.3;
      =     M   7002.7;
      A     L      0.1;
      BLD   102;
      L     S5T#0MS;
      SD    T    723;
      A     L      0.0;
      A(    ;
      O     DB327.DBX 1073.3;
      O     ;
      A     M   7003.0;
      AN    I      0.1;
      AN    I     80.1;
      )     ;
      =     L      0.1;
      A     L      0.1;
      A     T    724;
      AN    M      3.3;
      =     M   7003.0;
      A     L      0.1;
      BLD   102;
      L     S5T#0MS;
      SD    T    724;
      A     L      0.0;
      A(    ;
      O     DB327.DBX 1075.3;
      O     ;
      A     M   7003.1;
      AN    I      0.1;
      AN    I     80.1;
      )     ;
      =     L      0.1;
      A     L      0.1;
      A     T    725;
      AN    M      3.3;
      =     M   7003.1;
      A     L      0.1;
      BLD   102;
      L     S5T#0MS;
      SD    T    725;
      A     L      0.0;
      A(    ;
      O     DB327.DBX 1077.3;
      O     ;
      A     M   7003.2;
      AN    I      0.1;
      AN    I     80.1;
      )     ;
      =     L      0.1;
      A     L      0.1;
      A     T    726;
      AN    M      3.3;
      =     M   7003.2;
      A     L      0.1;
      BLD   102;
      L     S5T#0MS;
      SD    T    726;
      A     L      0.0;
      A(    ;
      O     DB327.DBX 1079.3;
      O     ;
      A     M   7003.3;
      AN    I      0.1;
      AN    I     80.1;
      )     ;
      =     L      0.1;
      A     L      0.1;
      A     T    727;
      AN    M      3.3;
      =     M   7003.3;
      A     L      0.1;
      BLD   102;
      L     S5T#0MS;
      SD    T    727;
      A     L      0.0;
      A(    ;
      O     DB327.DBX 1081.3;
      O     ;
      A     M   7003.4;
      AN    I      0.1;
      AN    I     80.1;
      )     ;
      =     L      0.1;
      A     L      0.1;
      A     T    728;
      AN    M      3.3;
      =     M   7003.4;
      A     L      0.1;
      BLD   102;
      L     S5T#0MS;
      SD    T    728;
      A     L      0.0;
      A(    ;
      O     DB327.DBX 1083.3;
      O     ;
      A     M   7003.5;
      AN    I      0.1;
      AN    I     80.1;
      )     ;
      =     L      0.1;
      A     L      0.1;
      A     T    729;
      AN    M      3.3;
      =     M   7003.5;
      A     L      0.1;
      BLD   102;
      L     S5T#0MS;
      SD    T    729;
NETWORK
TITLE =PROFINET ERROR(31~40)
//
//
      A     M      3.3;
      =     L      0.0;
      A     L      0.0;
      A(    ;
      O     DB327.DBX 1085.3;
      O     ;
      A     M   7003.6;
      AN    I      0.1;
      AN    I     80.1;
      )     ;
      =     L      0.1;
      A     L      0.1;
      A     T    730;
      AN    M      3.3;
      =     M   7003.6;
      A     L      0.1;
      BLD   102;
      L     S5T#0MS;
      SD    T    730;
      A     L      0.0;
      A(    ;
      O     DB327.DBX 1087.3;
      O     ;
      A     M   7003.7;
      AN    I      0.1;
      AN    I     80.1;
      )     ;
      =     L      0.1;
      A     L      0.1;
      A     T    731;
      AN    M      3.3;
      =     M   7003.7;
      A     L      0.1;
      BLD   102;
      L     S5T#0MS;
      SD    T    731;
      A     L      0.0;
      A(    ;
      O     DB327.DBX 1089.3;
      O     ;
      A     M   7004.0;
      AN    I      0.1;
      AN    I     80.1;
      )     ;
      =     L      0.1;
      A     L      0.1;
      A     T    732;
      AN    M      3.3;
      =     M   7004.0;
      A     L      0.1;
      BLD   102;
      L     S5T#0MS;
      SD    T    732;
      A     L      0.0;
      A(    ;
      O     DB327.DBX 1091.3;
      O     ;
      A     M   7004.1;
      AN    I      0.1;
      AN    I     80.1;
      )     ;
      =     L      0.1;
      A     L      0.1;
      A     T    733;
      AN    M      3.3;
      =     M   7004.1;
      A     L      0.1;
      BLD   102;
      L     S5T#0MS;
      SD    T    733;
      A     L      0.0;
      A(    ;
      O     DB327.DBX 1093.3;
      O     ;
      A     M   7004.2;
      AN    I      0.1;
      AN    I     80.1;
      )     ;
      =     L      0.1;
      A     L      0.1;
      A     T    734;
      AN    M      3.3;
      =     M   7004.2;
      A     L      0.1;
      BLD   102;
      L     S5T#0MS;
      SD    T    734;
      A     L      0.0;
      A(    ;
      O     DB327.DBX 1095.3;
      O     ;
      A     M   7004.3;
      AN    I      0.1;
      AN    I     80.1;
      )     ;
      =     L      0.1;
      A     L      0.1;
      A     T    735;
      AN    M      3.3;
      =     M   7004.3;
      A     L      0.1;
      BLD   102;
      L     S5T#0MS;
      SD    T    735;
      A     L      0.0;
      A(    ;
      O     DB327.DBX 1097.3;
      O     ;
      A     M   7004.4;
      AN    I      0.1;
      AN    I     80.1;
      )     ;
      =     L      0.1;
      A     L      0.1;
      A     T    736;
      AN    M      3.3;
      =     M   7004.4;
      A     L      0.1;
      BLD   102;
      L     S5T#0MS;
      SD    T    736;
      A     L      0.0;
      A(    ;
      O     DB327.DBX 1099.3;
      O     ;
      A     M   7004.5;
      AN    I      0.1;
      AN    I     80.1;
      )     ;
      =     L      0.1;
      A     L      0.1;
      A     T    737;
      AN    M      3.3;
      =     M   7004.5;
      A     L      0.1;
      BLD   102;
      L     S5T#0MS;
      SD    T    737;
      A     L      0.0;
      A(    ;
      O     DB327.DBX 1101.3;
      O     ;
      A     M   7004.6;
      AN    I      0.1;
      AN    I     80.1;
      )     ;
      =     L      0.1;
      A     L      0.1;
      A     T    738;
      AN    M      3.3;
      =     M   7004.6;
      A     L      0.1;
      BLD   102;
      L     S5T#0MS;
      SD    T    738;
      A     L      0.0;
      A(    ;
      O     DB327.DBX 1103.3;
      O     ;
      A     M   7004.7;
      AN    I      0.1;
      AN    I     80.1;
      )     ;
      =     L      0.1;
      A     L      0.1;
      A     T    739;
      AN    M      3.3;
      =     M   7004.7;
      A     L      0.1;
      BLD   102;
      L     S5T#0MS;
      SD    T    739;
NETWORK
TITLE =PROFINET ERROR(150~159)

      A     M      3.3;
      =     L      0.0;
      A     L      0.0;
      A(    ;
      O     DB327.DBX 1323.3;
      O     ;
      A     M   7018.5;
      AN    I      0.1;
      AN    I     80.1;
      )     ;
      =     L      0.1;
      A     L      0.1;
      A     T    849;
      =     M   7018.5;
      A     L      0.1;
      BLD   102;
      L     S5T#0MS;
      SD    T    849;
      A     L      0.0;
      A(    ;
      O     DB327.DBX 1325.3;
      O     ;
      A     M   7018.6;
      AN    I      0.1;
      AN    I     80.1;
      )     ;
      =     L      0.1;
      A     L      0.1;
      A     T    850;
      AN    M      3.3;
      =     M   7018.6;
      A     L      0.1;
      BLD   102;
      L     S5T#0MS;
      SD    T    850;
      A     L      0.0;
      A(    ;
      O     DB327.DBX 1327.3;
      O     ;
      A     M   7018.7;
      AN    I      0.1;
      AN    I     80.1;
      )     ;
      =     L      0.1;
      A     L      0.1;
      A     T    851;
      AN    M      3.3;
      =     M   7018.7;
      A     L      0.1;
      BLD   102;
      L     S5T#0MS;
      SD    T    851;
      A     L      0.0;
      A(    ;
      O     DB327.DBX 1329.3;
      O     ;
      A     M   7019.0;
      AN    I      0.1;
      AN    I     80.1;
      )     ;
      =     L      0.1;
      A     L      0.1;
      A     T    852;
      AN    M      3.3;
      =     M   7019.0;
      A     L      0.1;
      BLD   102;
      L     S5T#0MS;
      SD    T    852;
      A     L      0.0;
      A(    ;
      O     DB327.DBX 1331.3;
      O     ;
      A     M   7019.1;
      AN    I      0.1;
      AN    I     80.1;
      )     ;
      =     L      0.1;
      A     L      0.1;
      A     T    853;
      AN    M      3.3;
      =     M   7019.1;
      A     L      0.1;
      BLD   102;
      L     S5T#0MS;
      SD    T    853;
      A     L      0.0;
      A(    ;
      O     DB327.DBX 1333.3;
      O     ;
      A     M   7019.2;
      AN    I      0.1;
      AN    I     80.1;
      )     ;
      =     L      0.1;
      A     L      0.1;
      A     T    854;
      AN    M      3.3;
      =     M   7019.2;
      A     L      0.1;
      BLD   102;
      L     S5T#0MS;
      SD    T    854;
      A     L      0.0;
      A(    ;
      O     DB327.DBX 1335.3;
      O     ;
      A     M   7019.3;
      AN    I      0.1;
      AN    I     80.1;
      )     ;
      =     L      0.1;
      A     L      0.1;
      A     T    855;
      AN    M      3.3;
      =     M   7019.3;
      A     L      0.1;
      BLD   102;
      L     S5T#0MS;
      SD    T    855;
      A     L      0.0;
      A(    ;
      O     DB327.DBX 1337.3;
      O     ;
      A     M   7019.4;
      AN    I      0.1;
      AN    I     80.1;
      )     ;
      =     L      0.1;
      A     L      0.1;
      A     T    856;
      AN    M      3.3;
      =     M   7019.4;
      A     L      0.1;
      BLD   102;
      L     S5T#0MS;
      SD    T    856;
      A     L      0.0;
      A(    ;
      O     DB327.DBX 1339.3;
      O     ;
      A     M   7019.5;
      AN    I      0.1;
      AN    I     80.1;
      )     ;
      =     L      0.1;
      A     L      0.1;
      A     T    857;
      AN    M      3.3;
      =     M   7019.5;
      A     L      0.1;
      BLD   102;
      L     S5T#0MS;
      SD    T    857;
      A     L      0.0;
      A(    ;
      O     DB327.DBX 1341.3;
      O     ;
      A     M   7019.6;
      AN    I      0.1;
      AN    I     80.1;
      )     ;
      =     L      0.1;
      A     L      0.1;
      A     T    858;
      AN    M      3.3;
      =     M   7019.6;
      A     L      0.1;
      BLD   102;
      L     S5T#0MS;
      SD    T    858;
NETWORK
TITLE =CP TRIP(20~29)
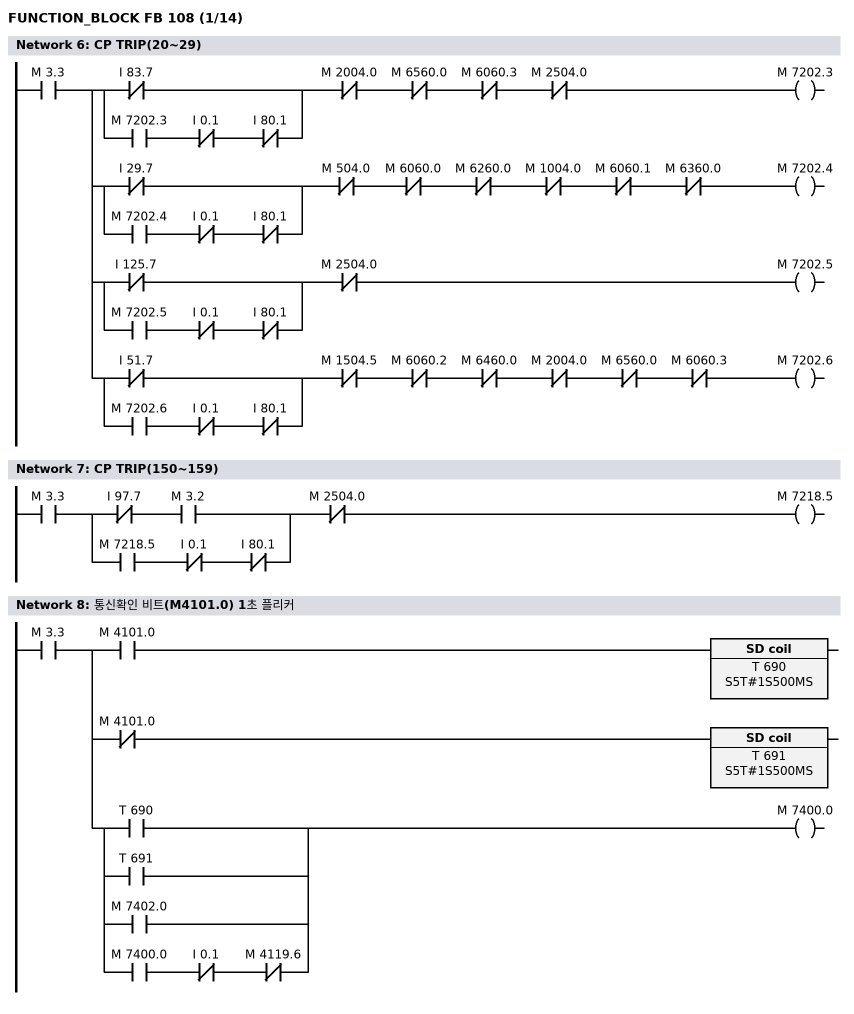

      A     M      3.3;
      =     L      0.0;
      A     L      0.0;
      A(    ;
      ON    I     83.7;
      O     ;
      A     M   7202.3;
      AN    I      0.1;
      AN    I     80.1;
      )     ;
      AN    M   2004.0;
      AN    M   6560.0;
      AN    M   6060.3;
      AN    M   2504.0;
      =     M   7202.3;
      A     L      0.0;
      A(    ;
      ON    I     29.7;
      O     ;
      A     M   7202.4;
      AN    I      0.1;
      AN    I     80.1;
      )     ;
      AN    M    504.0;
      AN    M   6060.0;
      AN    M   6260.0;
      AN    M   1004.0;
      AN    M   6060.1;
      AN    M   6360.0;
      =     M   7202.4;
      A     L      0.0;
      A(    ;
      ON    I    125.7;
      O     ;
      A     M   7202.5;
      AN    I      0.1;
      AN    I     80.1;
      )     ;
      AN    M   2504.0;
      =     M   7202.5;
      A     L      0.0;
      A(    ;
      ON    I     51.7;
      O     ;
      A     M   7202.6;
      AN    I      0.1;
      AN    I     80.1;
      )     ;
      AN    M   1504.5;
      AN    M   6060.2;
      AN    M   6460.0;
      AN    M   2004.0;
      AN    M   6560.0;
      AN    M   6060.3;
      =     M   7202.6;
NETWORK
TITLE =CP TRIP(150~159)

      A     M      3.3;
      A(    ;
      AN    I     97.7;
      A     M      3.2;
      O     ;
      A     M   7218.5;
      AN    I      0.1;
      AN    I     80.1;
      )     ;
      AN    M   2504.0;
      =     M   7218.5;
NETWORK
TITLE =통신확인 비트(M4101.0) 1초 플리커
//
//
//
      A     M      3.3;
      =     L      0.0;
      A     L      0.0;
      A     M   4101.0;
      L     S5T#1S500MS;
      SD    T    690;
      A     L      0.0;
      AN    M   4101.0;
      L     S5T#1S500MS;
      SD    T    691;
      A     L      0.0;
      A(    ;
      O     T    690;
      O     T    691;
      O     M   7402.0;
      O     ;
      A     M   7400.0;
      AN    I      0.1;
      AN    M   4119.6;
      )     ;
      =     M   7400.0;
NETWORK
TITLE =통신확인 비트(M5601.0) 1초 플리커
//
//
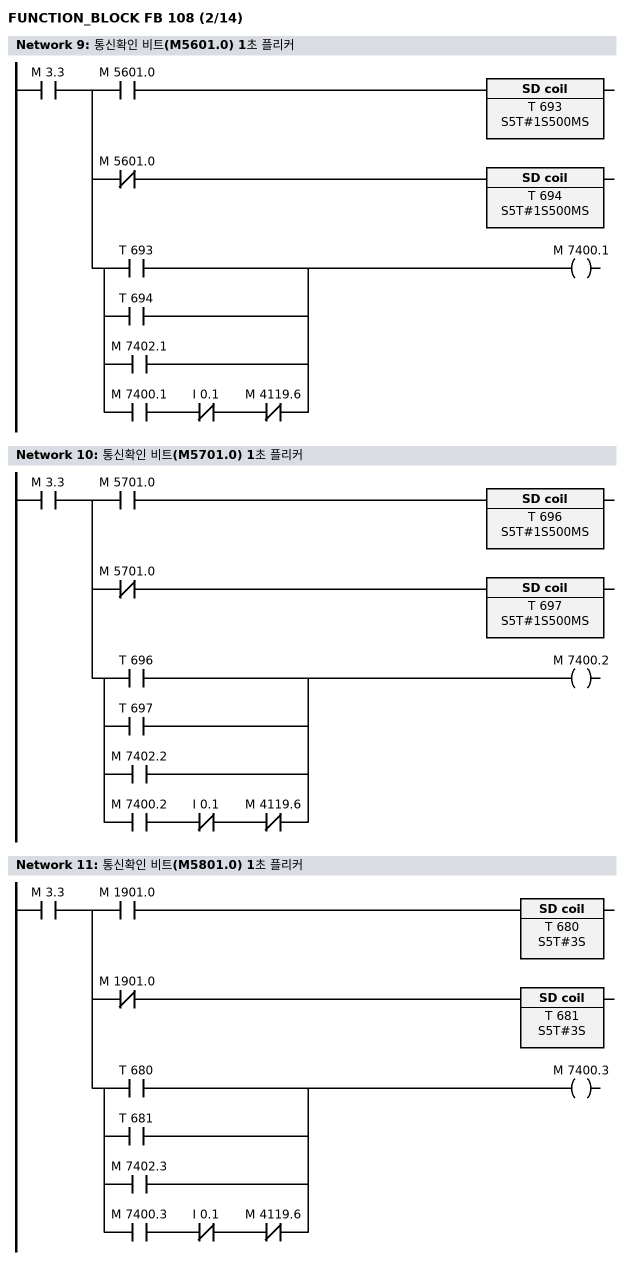
      A     M      3.3;
      =     L      0.0;
      A     L      0.0;
      A     M   5601.0;
      L     S5T#1S500MS;
      SD    T    693;
      A     L      0.0;
      AN    M   5601.0;
      L     S5T#1S500MS;
      SD    T    694;
      A     L      0.0;
      A(    ;
      O     T    693;
      O     T    694;
      O     M   7402.1;
      O     ;
      A     M   7400.1;
      AN    I      0.1;
      AN    M   4119.6;
      )     ;
      =     M   7400.1;
NETWORK
TITLE =통신확인 비트(M5701.0) 1초 플리커
//
//
      A     M      3.3;
      =     L      0.0;
      A     L      0.0;
      A     M   5701.0;
      L     S5T#1S500MS;
      SD    T    696;
      A     L      0.0;
      AN    M   5701.0;
      L     S5T#1S500MS;
      SD    T    697;
      A     L      0.0;
      A(    ;
      O     T    696;
      O     T    697;
      O     M   7402.2;
      O     ;
      A     M   7400.2;
      AN    I      0.1;
      AN    M   4119.6;
      )     ;
      =     M   7400.2;
NETWORK
TITLE =통신확인 비트(M5801.0) 1초 플리커
//
//
      A     M      3.3;
      =     L      0.0;
      A     L      0.0;
      A     M   1901.0;
      L     S5T#3S;
      SD    T    680;
      A     L      0.0;
      AN    M   1901.0;
      L     S5T#3S;
      SD    T    681;
      A     L      0.0;
      A(    ;
      O     T    680;
      O     T    681;
      O     M   7402.3;
      O     ;
      A     M   7400.3;
      AN    I      0.1;
      AN    M   4119.6;
      )     ;
      =     M   7400.3;
NETWORK
TITLE =제어반 허브1 알람
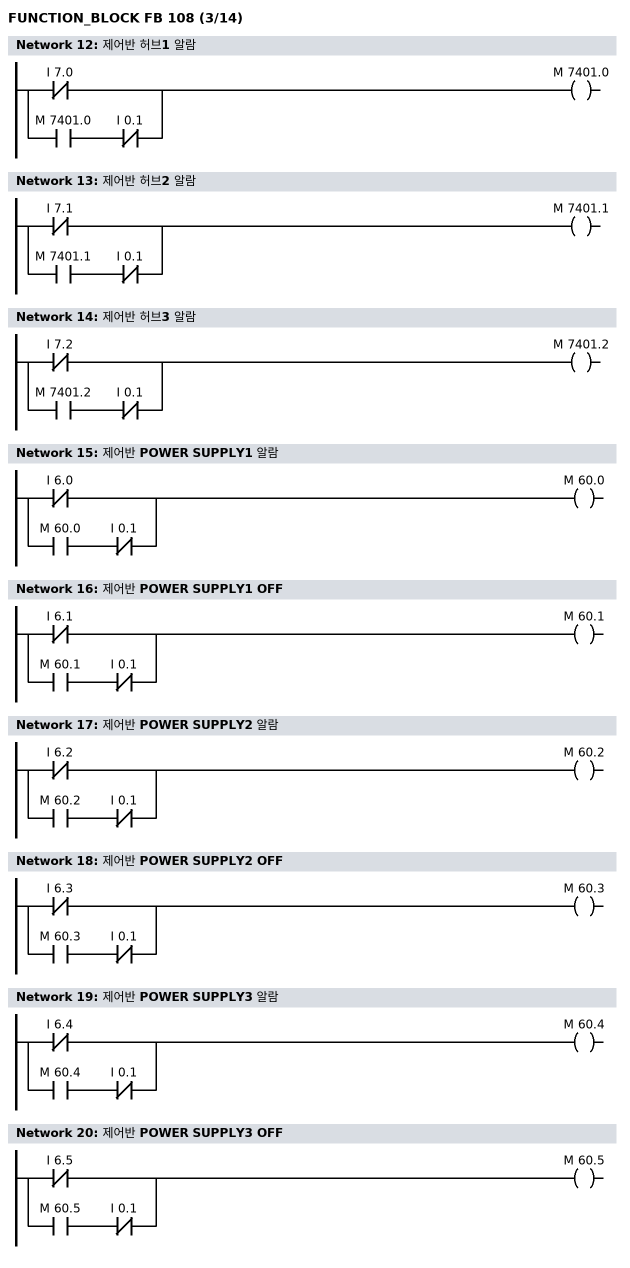

      ON    I      7.0;
      O     ;
      A     M   7401.0;
      AN    I      0.1;
      =     M   7401.0;
NETWORK
TITLE =제어반 허브2 알람

      ON    I      7.1;
      O     ;
      A     M   7401.1;
      AN    I      0.1;
      =     M   7401.1;
NETWORK
TITLE =제어반 허브3 알람

      ON    I      7.2;
      O     ;
      A     M   7401.2;
      AN    I      0.1;
      =     M   7401.2;
NETWORK
TITLE =제어반 POWER SUPPLY1 알람

      ON    I      6.0;
      O     ;
      A     M     60.0;
      AN    I      0.1;
      =     M     60.0;
NETWORK
TITLE =제어반 POWER SUPPLY1 OFF

      ON    I      6.1;
      O     ;
      A     M     60.1;
      AN    I      0.1;
      =     M     60.1;
NETWORK
TITLE =제어반 POWER SUPPLY2 알람
//
//
      ON    I      6.2;
      O     ;
      A     M     60.2;
      AN    I      0.1;
      =     M     60.2;
NETWORK
TITLE =제어반 POWER SUPPLY2 OFF

      ON    I      6.3;
      O     ;
      A     M     60.3;
      AN    I      0.1;
      =     M     60.3;
NETWORK
TITLE =제어반 POWER SUPPLY3 알람
//
//
      ON    I      6.4;
      O     ;
      A     M     60.4;
      AN    I      0.1;
      =     M     60.4;
NETWORK
TITLE =제어반 POWER SUPPLY3 OFF

      ON    I      6.5;
      O     ;
      A     M     60.5;
      AN    I      0.1;
      =     M     60.5;
NETWORK
TITLE =제어반 서지보호기 알람
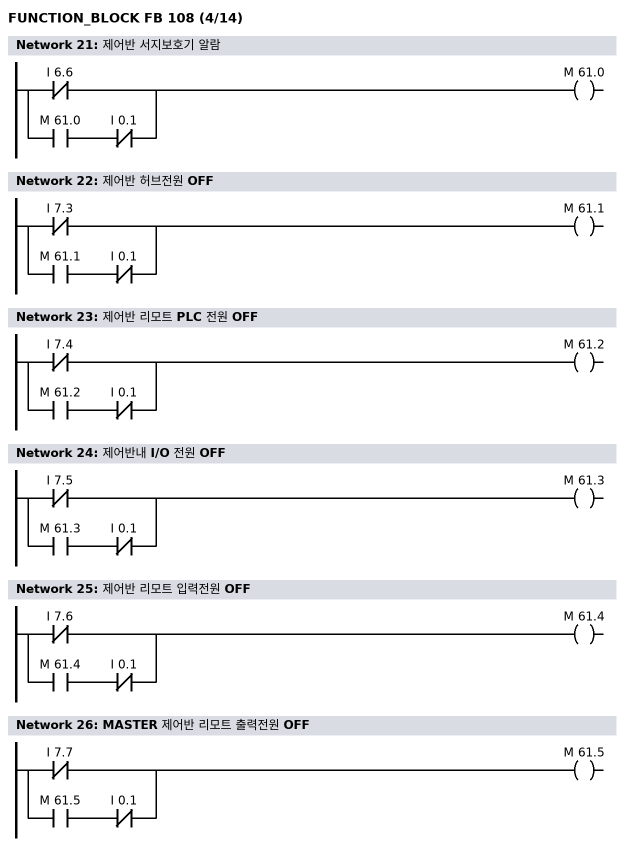

      ON    I      6.6;
      O     ;
      A     M     61.0;
      AN    I      0.1;
      =     M     61.0;
NETWORK
TITLE =제어반 허브전원 OFF

      ON    I      7.3;
      O     ;
      A     M     61.1;
      AN    I      0.1;
      =     M     61.1;
NETWORK
TITLE =제어반 리모트 PLC 전원 OFF

      ON    I      7.4;
      O     ;
      A     M     61.2;
      AN    I      0.1;
      =     M     61.2;
NETWORK
TITLE =제어반내 I/O 전원 OFF

      ON    I      7.5;
      O     ;
      A     M     61.3;
      AN    I      0.1;
      =     M     61.3;
NETWORK
TITLE =제어반 리모트 입력전원 OFF

      ON    I      7.6;
      O     ;
      A     M     61.4;
      AN    I      0.1;
      =     M     61.4;
NETWORK
TITLE =MASTER 제어반 리모트 출력전원 OFF

      ON    I      7.7;
      O     ;
      A     M     61.5;
      AN    I      0.1;
      =     M     61.5;
NETWORK
TITLE =PROFINET ALARM-모듈이상이나 통신케이블단선(1~10)
//
//
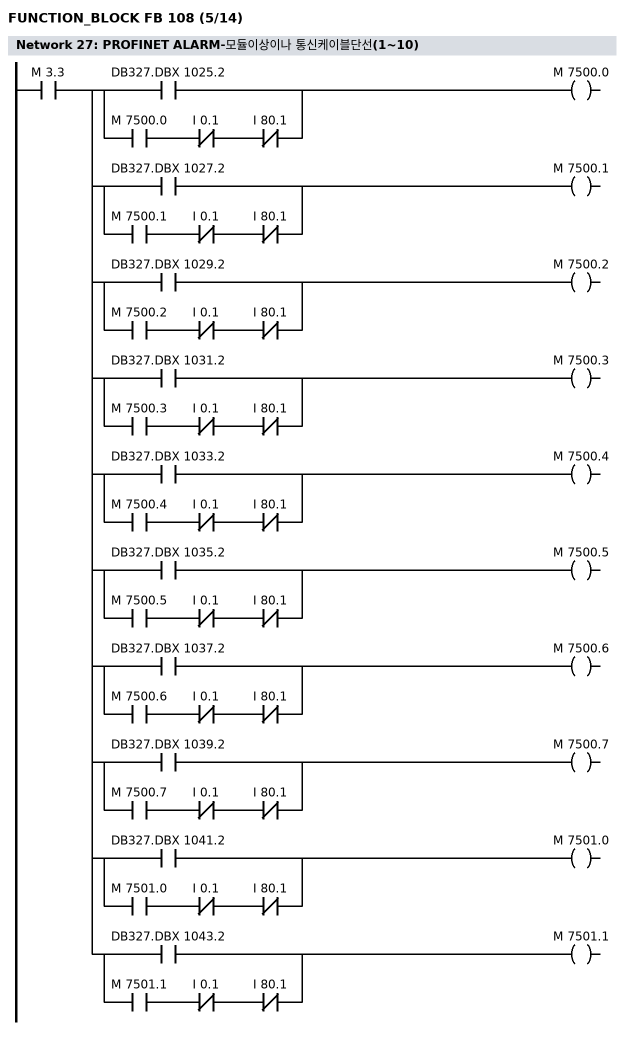
      A     M      3.3;
      =     L      0.0;
      A     L      0.0;
      A(    ;
      O     DB327.DBX 1025.2;
      O     ;
      A     M   7500.0;
      AN    I      0.1;
      AN    I     80.1;
      )     ;
      =     M   7500.0;
      A     L      0.0;
      A(    ;
      O     DB327.DBX 1027.2;
      O     ;
      A     M   7500.1;
      AN    I      0.1;
      AN    I     80.1;
      )     ;
      =     M   7500.1;
      A     L      0.0;
      A(    ;
      O     DB327.DBX 1029.2;
      O     ;
      A     M   7500.2;
      AN    I      0.1;
      AN    I     80.1;
      )     ;
      =     M   7500.2;
      A     L      0.0;
      A(    ;
      O     DB327.DBX 1031.2;
      O     ;
      A     M   7500.3;
      AN    I      0.1;
      AN    I     80.1;
      )     ;
      =     M   7500.3;
      A     L      0.0;
      A(    ;
      O     DB327.DBX 1033.2;
      O     ;
      A     M   7500.4;
      AN    I      0.1;
      AN    I     80.1;
      )     ;
      =     M   7500.4;
      A     L      0.0;
      A(    ;
      O     DB327.DBX 1035.2;
      O     ;
      A     M   7500.5;
      AN    I      0.1;
      AN    I     80.1;
      )     ;
      =     M   7500.5;
      A     L      0.0;
      A(    ;
      O     DB327.DBX 1037.2;
      O     ;
      A     M   7500.6;
      AN    I      0.1;
      AN    I     80.1;
      )     ;
      =     M   7500.6;
      A     L      0.0;
      A(    ;
      O     DB327.DBX 1039.2;
      O     ;
      A     M   7500.7;
      AN    I      0.1;
      AN    I     80.1;
      )     ;
      =     M   7500.7;
      A     L      0.0;
      A(    ;
      O     DB327.DBX 1041.2;
      O     ;
      A     M   7501.0;
      AN    I      0.1;
      AN    I     80.1;
      )     ;
      =     M   7501.0;
      A     L      0.0;
      A(    ;
      O     DB327.DBX 1043.2;
      O     ;
      A     M   7501.1;
      AN    I      0.1;
      AN    I     80.1;
      )     ;
      =     M   7501.1;
NETWORK
TITLE =PROFINET ALARM-모듈이상이나 통신케이블단선(11~20)
//
//
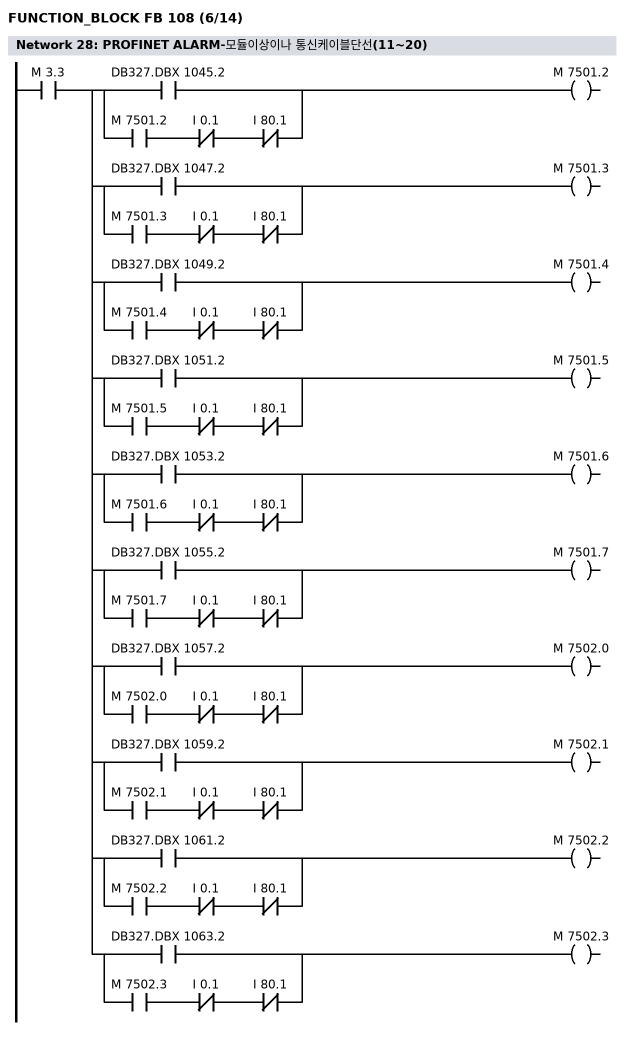
      A     M      3.3;
      =     L      0.0;
      A     L      0.0;
      A(    ;
      O     DB327.DBX 1045.2;
      O     ;
      A     M   7501.2;
      AN    I      0.1;
      AN    I     80.1;
      )     ;
      =     M   7501.2;
      A     L      0.0;
      A(    ;
      O     DB327.DBX 1047.2;
      O     ;
      A     M   7501.3;
      AN    I      0.1;
      AN    I     80.1;
      )     ;
      =     M   7501.3;
      A     L      0.0;
      A(    ;
      O     DB327.DBX 1049.2;
      O     ;
      A     M   7501.4;
      AN    I      0.1;
      AN    I     80.1;
      )     ;
      =     M   7501.4;
      A     L      0.0;
      A(    ;
      O     DB327.DBX 1051.2;
      O     ;
      A     M   7501.5;
      AN    I      0.1;
      AN    I     80.1;
      )     ;
      =     M   7501.5;
      A     L      0.0;
      A(    ;
      O     DB327.DBX 1053.2;
      O     ;
      A     M   7501.6;
      AN    I      0.1;
      AN    I     80.1;
      )     ;
      =     M   7501.6;
      A     L      0.0;
      A(    ;
      O     DB327.DBX 1055.2;
      O     ;
      A     M   7501.7;
      AN    I      0.1;
      AN    I     80.1;
      )     ;
      =     M   7501.7;
      A     L      0.0;
      A(    ;
      O     DB327.DBX 1057.2;
      O     ;
      A     M   7502.0;
      AN    I      0.1;
      AN    I     80.1;
      )     ;
      =     M   7502.0;
      A     L      0.0;
      A(    ;
      O     DB327.DBX 1059.2;
      O     ;
      A     M   7502.1;
      AN    I      0.1;
      AN    I     80.1;
      )     ;
      =     M   7502.1;
      A     L      0.0;
      A(    ;
      O     DB327.DBX 1061.2;
      O     ;
      A     M   7502.2;
      AN    I      0.1;
      AN    I     80.1;
      )     ;
      =     M   7502.2;
      A     L      0.0;
      A(    ;
      O     DB327.DBX 1063.2;
      O     ;
      A     M   7502.3;
      AN    I      0.1;
      AN    I     80.1;
      )     ;
      =     M   7502.3;
NETWORK
TITLE =PROFINET ALARM-모듈이상이나 통신케이블단선(21~30)
//
//
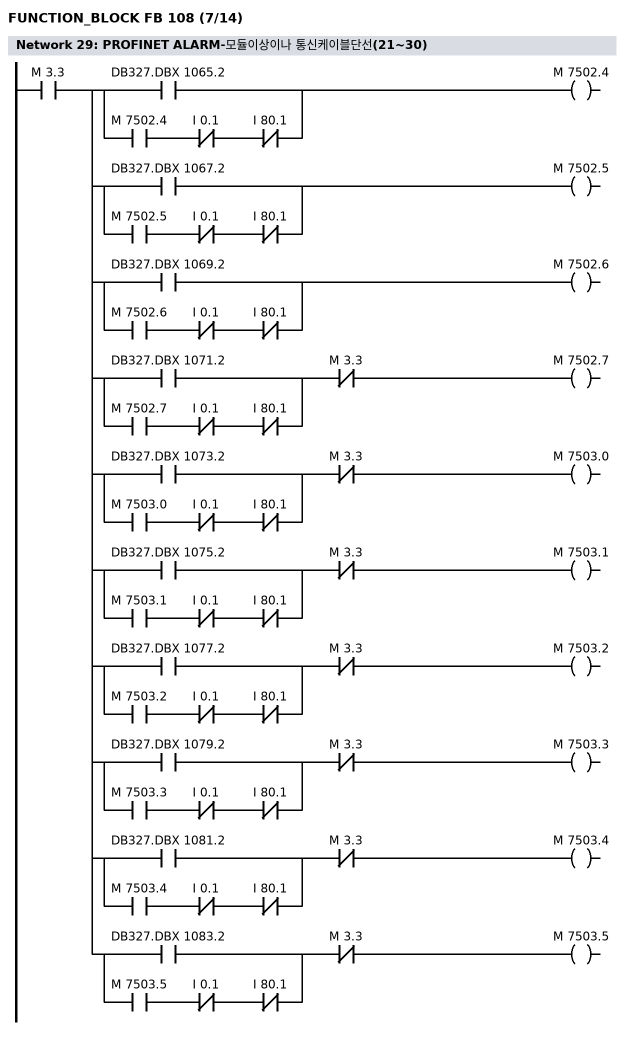
      A     M      3.3;
      =     L      0.0;
      A     L      0.0;
      A(    ;
      O     DB327.DBX 1065.2;
      O     ;
      A     M   7502.4;
      AN    I      0.1;
      AN    I     80.1;
      )     ;
      =     M   7502.4;
      A     L      0.0;
      A(    ;
      O     DB327.DBX 1067.2;
      O     ;
      A     M   7502.5;
      AN    I      0.1;
      AN    I     80.1;
      )     ;
      =     M   7502.5;
      A     L      0.0;
      A(    ;
      O     DB327.DBX 1069.2;
      O     ;
      A     M   7502.6;
      AN    I      0.1;
      AN    I     80.1;
      )     ;
      =     M   7502.6;
      A     L      0.0;
      A(    ;
      O     DB327.DBX 1071.2;
      O     ;
      A     M   7502.7;
      AN    I      0.1;
      AN    I     80.1;
      )     ;
      AN    M      3.3;
      =     M   7502.7;
      A     L      0.0;
      A(    ;
      O     DB327.DBX 1073.2;
      O     ;
      A     M   7503.0;
      AN    I      0.1;
      AN    I     80.1;
      )     ;
      AN    M      3.3;
      =     M   7503.0;
      A     L      0.0;
      A(    ;
      O     DB327.DBX 1075.2;
      O     ;
      A     M   7503.1;
      AN    I      0.1;
      AN    I     80.1;
      )     ;
      AN    M      3.3;
      =     M   7503.1;
      A     L      0.0;
      A(    ;
      O     DB327.DBX 1077.2;
      O     ;
      A     M   7503.2;
      AN    I      0.1;
      AN    I     80.1;
      )     ;
      AN    M      3.3;
      =     M   7503.2;
      A     L      0.0;
      A(    ;
      O     DB327.DBX 1079.2;
      O     ;
      A     M   7503.3;
      AN    I      0.1;
      AN    I     80.1;
      )     ;
      AN    M      3.3;
      =     M   7503.3;
      A     L      0.0;
      A(    ;
      O     DB327.DBX 1081.2;
      O     ;
      A     M   7503.4;
      AN    I      0.1;
      AN    I     80.1;
      )     ;
      AN    M      3.3;
      =     M   7503.4;
      A     L      0.0;
      A(    ;
      O     DB327.DBX 1083.2;
      O     ;
      A     M   7503.5;
      AN    I      0.1;
      AN    I     80.1;
      )     ;
      AN    M      3.3;
      =     M   7503.5;
NETWORK
TITLE =PROFINET ALARM-모듈이상이나 통신케이블단선(31~40)
//
//
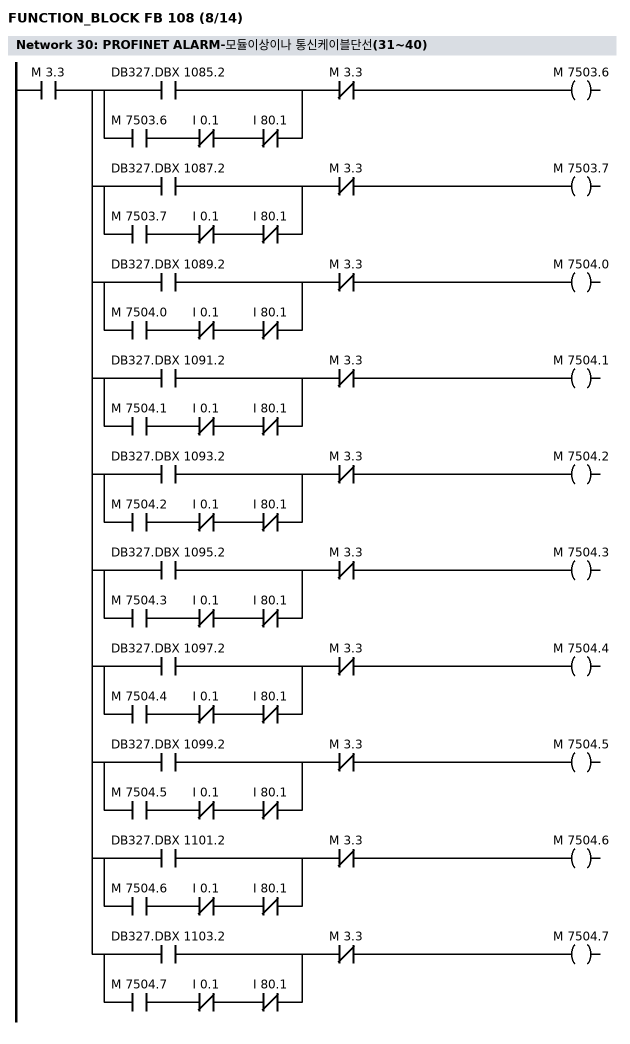
      A     M      3.3;
      =     L      0.0;
      A     L      0.0;
      A(    ;
      O     DB327.DBX 1085.2;
      O     ;
      A     M   7503.6;
      AN    I      0.1;
      AN    I     80.1;
      )     ;
      AN    M      3.3;
      =     M   7503.6;
      A     L      0.0;
      A(    ;
      O     DB327.DBX 1087.2;
      O     ;
      A     M   7503.7;
      AN    I      0.1;
      AN    I     80.1;
      )     ;
      AN    M      3.3;
      =     M   7503.7;
      A     L      0.0;
      A(    ;
      O     DB327.DBX 1089.2;
      O     ;
      A     M   7504.0;
      AN    I      0.1;
      AN    I     80.1;
      )     ;
      AN    M      3.3;
      =     M   7504.0;
      A     L      0.0;
      A(    ;
      O     DB327.DBX 1091.2;
      O     ;
      A     M   7504.1;
      AN    I      0.1;
      AN    I     80.1;
      )     ;
      AN    M      3.3;
      =     M   7504.1;
      A     L      0.0;
      A(    ;
      O     DB327.DBX 1093.2;
      O     ;
      A     M   7504.2;
      AN    I      0.1;
      AN    I     80.1;
      )     ;
      AN    M      3.3;
      =     M   7504.2;
      A     L      0.0;
      A(    ;
      O     DB327.DBX 1095.2;
      O     ;
      A     M   7504.3;
      AN    I      0.1;
      AN    I     80.1;
      )     ;
      AN    M      3.3;
      =     M   7504.3;
      A     L      0.0;
      A(    ;
      O     DB327.DBX 1097.2;
      O     ;
      A     M   7504.4;
      AN    I      0.1;
      AN    I     80.1;
      )     ;
      AN    M      3.3;
      =     M   7504.4;
      A     L      0.0;
      A(    ;
      O     DB327.DBX 1099.2;
      O     ;
      A     M   7504.5;
      AN    I      0.1;
      AN    I     80.1;
      )     ;
      AN    M      3.3;
      =     M   7504.5;
      A     L      0.0;
      A(    ;
      O     DB327.DBX 1101.2;
      O     ;
      A     M   7504.6;
      AN    I      0.1;
      AN    I     80.1;
      )     ;
      AN    M      3.3;
      =     M   7504.6;
      A     L      0.0;
      A(    ;
      O     DB327.DBX 1103.2;
      O     ;
      A     M   7504.7;
      AN    I      0.1;
      AN    I     80.1;
      )     ;
      AN    M      3.3;
      =     M   7504.7;
NETWORK
TITLE =PROFINET ALARM-모듈이상이나 통신케이블단선(150~159)
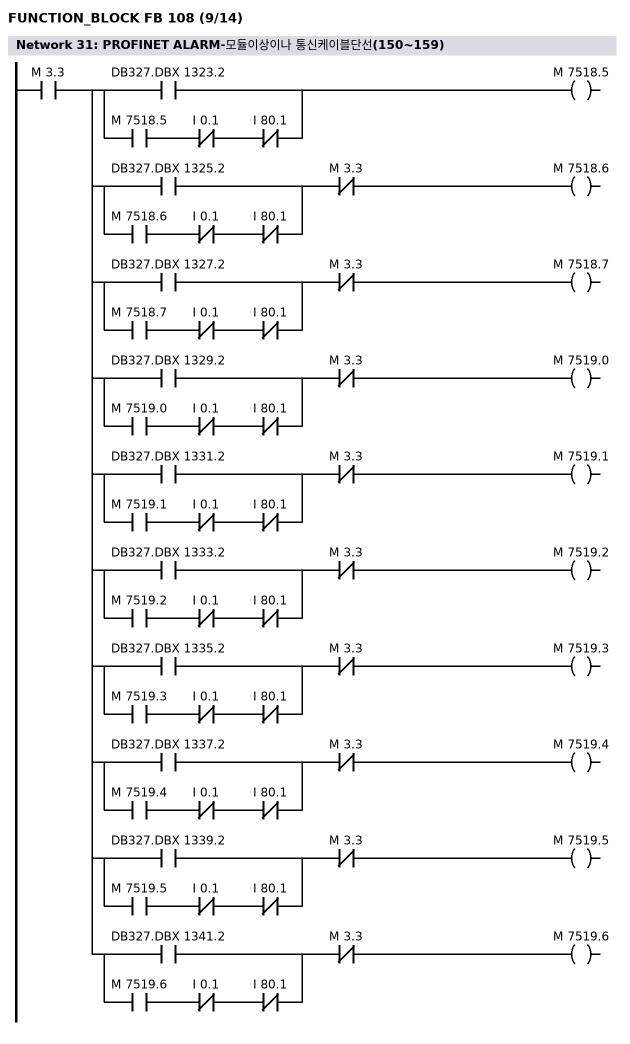

      A     M      3.3;
      =     L      0.0;
      A     L      0.0;
      A(    ;
      O     DB327.DBX 1323.2;
      O     ;
      A     M   7518.5;
      AN    I      0.1;
      AN    I     80.1;
      )     ;
      =     M   7518.5;
      A     L      0.0;
      A(    ;
      O     DB327.DBX 1325.2;
      O     ;
      A     M   7518.6;
      AN    I      0.1;
      AN    I     80.1;
      )     ;
      AN    M      3.3;
      =     M   7518.6;
      A     L      0.0;
      A(    ;
      O     DB327.DBX 1327.2;
      O     ;
      A     M   7518.7;
      AN    I      0.1;
      AN    I     80.1;
      )     ;
      AN    M      3.3;
      =     M   7518.7;
      A     L      0.0;
      A(    ;
      O     DB327.DBX 1329.2;
      O     ;
      A     M   7519.0;
      AN    I      0.1;
      AN    I     80.1;
      )     ;
      AN    M      3.3;
      =     M   7519.0;
      A     L      0.0;
      A(    ;
      O     DB327.DBX 1331.2;
      O     ;
      A     M   7519.1;
      AN    I      0.1;
      AN    I     80.1;
      )     ;
      AN    M      3.3;
      =     M   7519.1;
      A     L      0.0;
      A(    ;
      O     DB327.DBX 1333.2;
      O     ;
      A     M   7519.2;
      AN    I      0.1;
      AN    I     80.1;
      )     ;
      AN    M      3.3;
      =     M   7519.2;
      A     L      0.0;
      A(    ;
      O     DB327.DBX 1335.2;
      O     ;
      A     M   7519.3;
      AN    I      0.1;
      AN    I     80.1;
      )     ;
      AN    M      3.3;
      =     M   7519.3;
      A     L      0.0;
      A(    ;
      O     DB327.DBX 1337.2;
      O     ;
      A     M   7519.4;
      AN    I      0.1;
      AN    I     80.1;
      )     ;
      AN    M      3.3;
      =     M   7519.4;
      A     L      0.0;
      A(    ;
      O     DB327.DBX 1339.2;
      O     ;
      A     M   7519.5;
      AN    I      0.1;
      AN    I     80.1;
      )     ;
      AN    M      3.3;
      =     M   7519.5;
      A     L      0.0;
      A(    ;
      O     DB327.DBX 1341.2;
      O     ;
      A     M   7519.6;
      AN    I      0.1;
      AN    I     80.1;
      )     ;
      AN    M      3.3;
      =     M   7519.6;
NETWORK
TITLE =PROFINET MODULE ERROR(1~10)
//
//
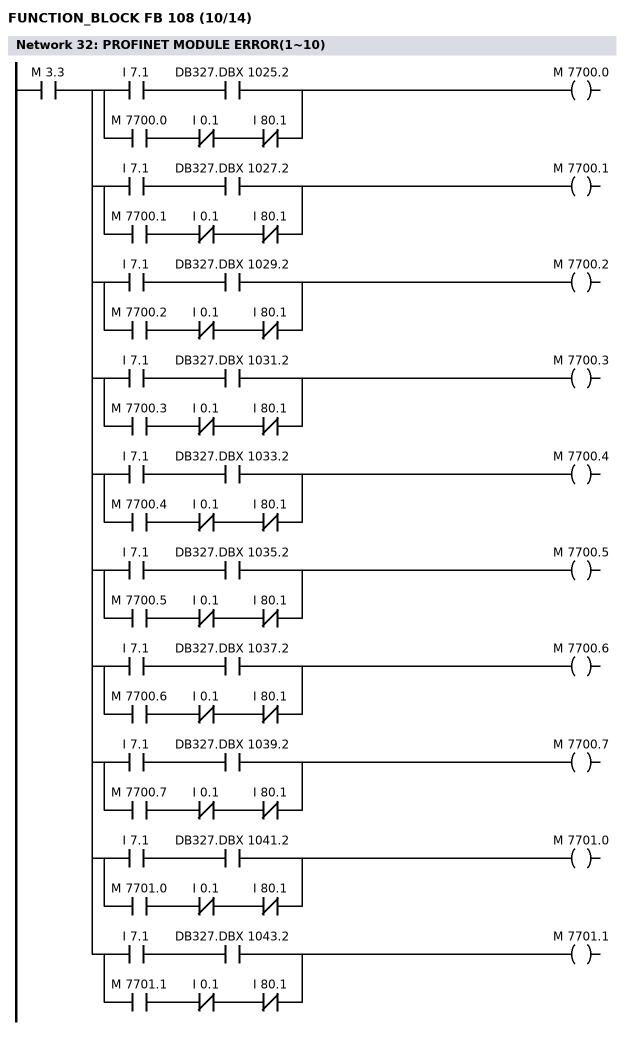
      A     M      3.3;
      =     L      0.0;
      A     L      0.0;
      A(    ;
      A     I      7.1;
      A     DB327.DBX 1025.2;
      O     ;
      A     M   7700.0;
      AN    I      0.1;
      AN    I     80.1;
      )     ;
      =     M   7700.0;
      A     L      0.0;
      A(    ;
      A     I      7.1;
      A     DB327.DBX 1027.2;
      O     ;
      A     M   7700.1;
      AN    I      0.1;
      AN    I     80.1;
      )     ;
      =     M   7700.1;
      A     L      0.0;
      A(    ;
      A     I      7.1;
      A     DB327.DBX 1029.2;
      O     ;
      A     M   7700.2;
      AN    I      0.1;
      AN    I     80.1;
      )     ;
      =     M   7700.2;
      A     L      0.0;
      A(    ;
      A     I      7.1;
      A     DB327.DBX 1031.2;
      O     ;
      A     M   7700.3;
      AN    I      0.1;
      AN    I     80.1;
      )     ;
      =     M   7700.3;
      A     L      0.0;
      A(    ;
      A     I      7.1;
      A     DB327.DBX 1033.2;
      O     ;
      A     M   7700.4;
      AN    I      0.1;
      AN    I     80.1;
      )     ;
      =     M   7700.4;
      A     L      0.0;
      A(    ;
      A     I      7.1;
      A     DB327.DBX 1035.2;
      O     ;
      A     M   7700.5;
      AN    I      0.1;
      AN    I     80.1;
      )     ;
      =     M   7700.5;
      A     L      0.0;
      A(    ;
      A     I      7.1;
      A     DB327.DBX 1037.2;
      O     ;
      A     M   7700.6;
      AN    I      0.1;
      AN    I     80.1;
      )     ;
      =     M   7700.6;
      A     L      0.0;
      A(    ;
      A     I      7.1;
      A     DB327.DBX 1039.2;
      O     ;
      A     M   7700.7;
      AN    I      0.1;
      AN    I     80.1;
      )     ;
      =     M   7700.7;
      A     L      0.0;
      A(    ;
      A     I      7.1;
      A     DB327.DBX 1041.2;
      O     ;
      A     M   7701.0;
      AN    I      0.1;
      AN    I     80.1;
      )     ;
      =     M   7701.0;
      A     L      0.0;
      A(    ;
      A     I      7.1;
      A     DB327.DBX 1043.2;
      O     ;
      A     M   7701.1;
      AN    I      0.1;
      AN    I     80.1;
      )     ;
      =     M   7701.1;
NETWORK
TITLE =PROFINET MODULE ERROR(11~20)
//
//
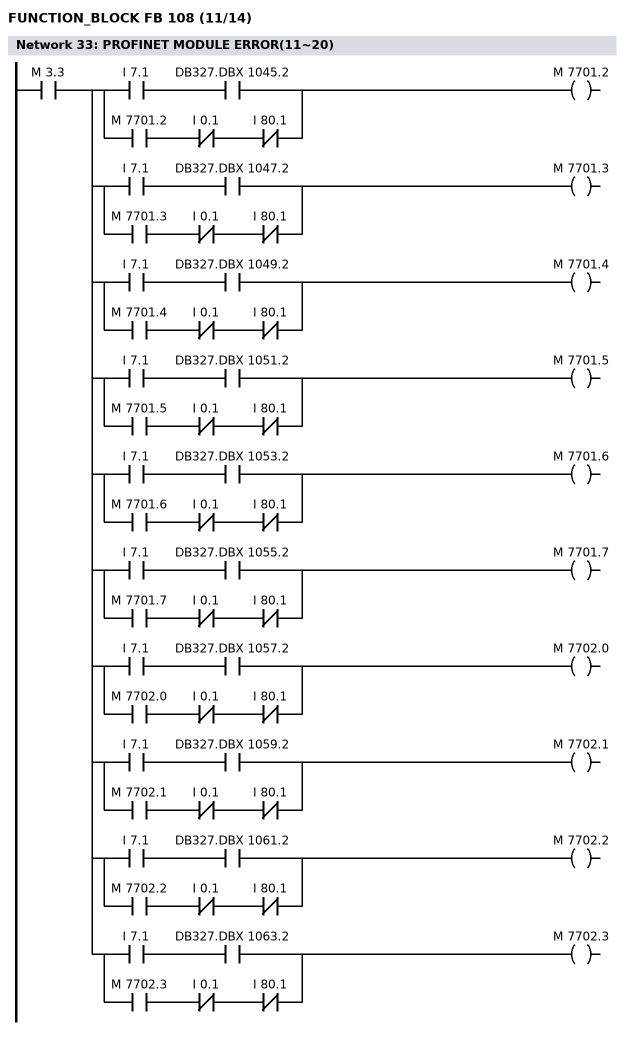
      A     M      3.3;
      =     L      0.0;
      A     L      0.0;
      A(    ;
      A     I      7.1;
      A     DB327.DBX 1045.2;
      O     ;
      A     M   7701.2;
      AN    I      0.1;
      AN    I     80.1;
      )     ;
      =     M   7701.2;
      A     L      0.0;
      A(    ;
      A     I      7.1;
      A     DB327.DBX 1047.2;
      O     ;
      A     M   7701.3;
      AN    I      0.1;
      AN    I     80.1;
      )     ;
      =     M   7701.3;
      A     L      0.0;
      A(    ;
      A     I      7.1;
      A     DB327.DBX 1049.2;
      O     ;
      A     M   7701.4;
      AN    I      0.1;
      AN    I     80.1;
      )     ;
      =     M   7701.4;
      A     L      0.0;
      A(    ;
      A     I      7.1;
      A     DB327.DBX 1051.2;
      O     ;
      A     M   7701.5;
      AN    I      0.1;
      AN    I     80.1;
      )     ;
      =     M   7701.5;
      A     L      0.0;
      A(    ;
      A     I      7.1;
      A     DB327.DBX 1053.2;
      O     ;
      A     M   7701.6;
      AN    I      0.1;
      AN    I     80.1;
      )     ;
      =     M   7701.6;
      A     L      0.0;
      A(    ;
      A     I      7.1;
      A     DB327.DBX 1055.2;
      O     ;
      A     M   7701.7;
      AN    I      0.1;
      AN    I     80.1;
      )     ;
      =     M   7701.7;
      A     L      0.0;
      A(    ;
      A     I      7.1;
      A     DB327.DBX 1057.2;
      O     ;
      A     M   7702.0;
      AN    I      0.1;
      AN    I     80.1;
      )     ;
      =     M   7702.0;
      A     L      0.0;
      A(    ;
      A     I      7.1;
      A     DB327.DBX 1059.2;
      O     ;
      A     M   7702.1;
      AN    I      0.1;
      AN    I     80.1;
      )     ;
      =     M   7702.1;
      A     L      0.0;
      A(    ;
      A     I      7.1;
      A     DB327.DBX 1061.2;
      O     ;
      A     M   7702.2;
      AN    I      0.1;
      AN    I     80.1;
      )     ;
      =     M   7702.2;
      A     L      0.0;
      A(    ;
      A     I      7.1;
      A     DB327.DBX 1063.2;
      O     ;
      A     M   7702.3;
      AN    I      0.1;
      AN    I     80.1;
      )     ;
      =     M   7702.3;
NETWORK
TITLE =PROFINET MODULE ERROR(21~30)
//
//
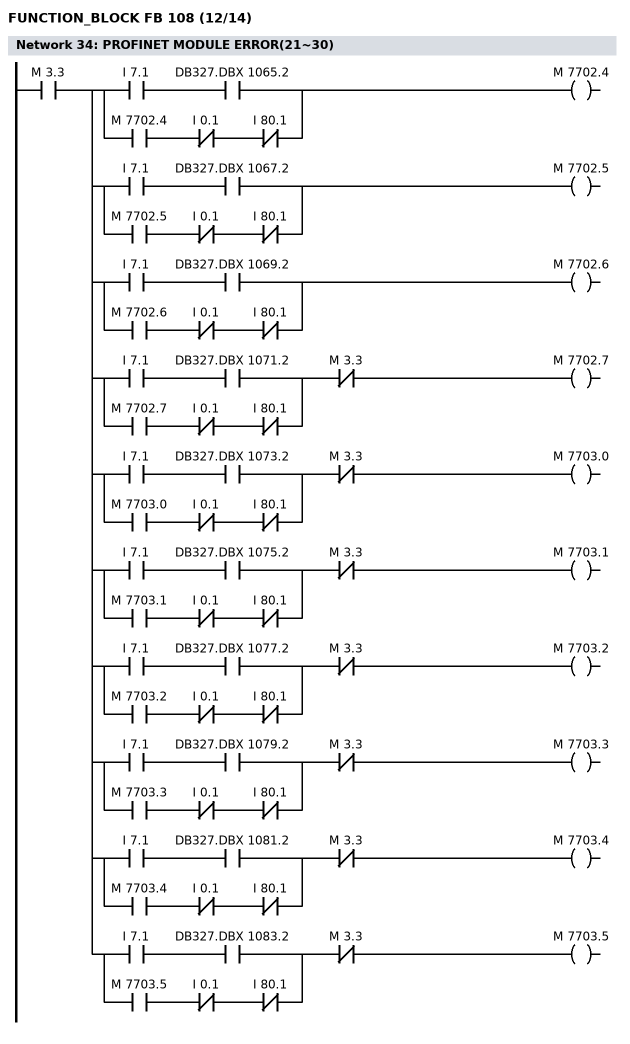
      A     M      3.3;
      =     L      0.0;
      A     L      0.0;
      A(    ;
      A     I      7.1;
      A     DB327.DBX 1065.2;
      O     ;
      A     M   7702.4;
      AN    I      0.1;
      AN    I     80.1;
      )     ;
      =     M   7702.4;
      A     L      0.0;
      A(    ;
      A     I      7.1;
      A     DB327.DBX 1067.2;
      O     ;
      A     M   7702.5;
      AN    I      0.1;
      AN    I     80.1;
      )     ;
      =     M   7702.5;
      A     L      0.0;
      A(    ;
      A     I      7.1;
      A     DB327.DBX 1069.2;
      O     ;
      A     M   7702.6;
      AN    I      0.1;
      AN    I     80.1;
      )     ;
      =     M   7702.6;
      A     L      0.0;
      A(    ;
      A     I      7.1;
      A     DB327.DBX 1071.2;
      O     ;
      A     M   7702.7;
      AN    I      0.1;
      AN    I     80.1;
      )     ;
      AN    M      3.3;
      =     M   7702.7;
      A     L      0.0;
      A(    ;
      A     I      7.1;
      A     DB327.DBX 1073.2;
      O     ;
      A     M   7703.0;
      AN    I      0.1;
      AN    I     80.1;
      )     ;
      AN    M      3.3;
      =     M   7703.0;
      A     L      0.0;
      A(    ;
      A     I      7.1;
      A     DB327.DBX 1075.2;
      O     ;
      A     M   7703.1;
      AN    I      0.1;
      AN    I     80.1;
      )     ;
      AN    M      3.3;
      =     M   7703.1;
      A     L      0.0;
      A(    ;
      A     I      7.1;
      A     DB327.DBX 1077.2;
      O     ;
      A     M   7703.2;
      AN    I      0.1;
      AN    I     80.1;
      )     ;
      AN    M      3.3;
      =     M   7703.2;
      A     L      0.0;
      A(    ;
      A     I      7.1;
      A     DB327.DBX 1079.2;
      O     ;
      A     M   7703.3;
      AN    I      0.1;
      AN    I     80.1;
      )     ;
      AN    M      3.3;
      =     M   7703.3;
      A     L      0.0;
      A(    ;
      A     I      7.1;
      A     DB327.DBX 1081.2;
      O     ;
      A     M   7703.4;
      AN    I      0.1;
      AN    I     80.1;
      )     ;
      AN    M      3.3;
      =     M   7703.4;
      A     L      0.0;
      A(    ;
      A     I      7.1;
      A     DB327.DBX 1083.2;
      O     ;
      A     M   7703.5;
      AN    I      0.1;
      AN    I     80.1;
      )     ;
      AN    M      3.3;
      =     M   7703.5;
NETWORK
TITLE =PROFINET MODULE ERROR(31~40)
//
//
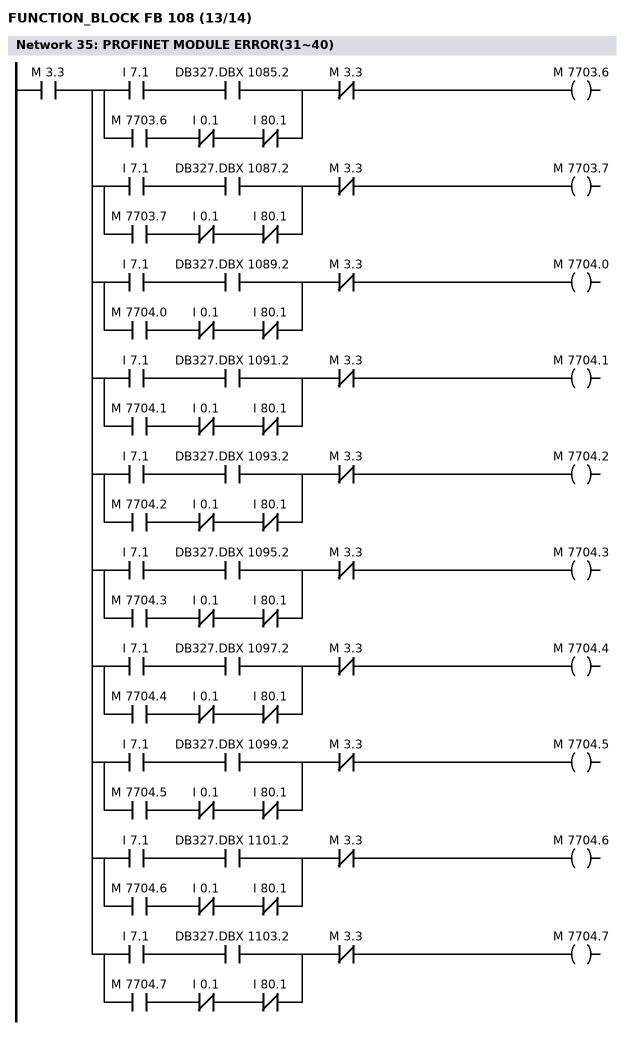
      A     M      3.3;
      =     L      0.0;
      A     L      0.0;
      A(    ;
      A     I      7.1;
      A     DB327.DBX 1085.2;
      O     ;
      A     M   7703.6;
      AN    I      0.1;
      AN    I     80.1;
      )     ;
      AN    M      3.3;
      =     M   7703.6;
      A     L      0.0;
      A(    ;
      A     I      7.1;
      A     DB327.DBX 1087.2;
      O     ;
      A     M   7703.7;
      AN    I      0.1;
      AN    I     80.1;
      )     ;
      AN    M      3.3;
      =     M   7703.7;
      A     L      0.0;
      A(    ;
      A     I      7.1;
      A     DB327.DBX 1089.2;
      O     ;
      A     M   7704.0;
      AN    I      0.1;
      AN    I     80.1;
      )     ;
      AN    M      3.3;
      =     M   7704.0;
      A     L      0.0;
      A(    ;
      A     I      7.1;
      A     DB327.DBX 1091.2;
      O     ;
      A     M   7704.1;
      AN    I      0.1;
      AN    I     80.1;
      )     ;
      AN    M      3.3;
      =     M   7704.1;
      A     L      0.0;
      A(    ;
      A     I      7.1;
      A     DB327.DBX 1093.2;
      O     ;
      A     M   7704.2;
      AN    I      0.1;
      AN    I     80.1;
      )     ;
      AN    M      3.3;
      =     M   7704.2;
      A     L      0.0;
      A(    ;
      A     I      7.1;
      A     DB327.DBX 1095.2;
      O     ;
      A     M   7704.3;
      AN    I      0.1;
      AN    I     80.1;
      )     ;
      AN    M      3.3;
      =     M   7704.3;
      A     L      0.0;
      A(    ;
      A     I      7.1;
      A     DB327.DBX 1097.2;
      O     ;
      A     M   7704.4;
      AN    I      0.1;
      AN    I     80.1;
      )     ;
      AN    M      3.3;
      =     M   7704.4;
      A     L      0.0;
      A(    ;
      A     I      7.1;
      A     DB327.DBX 1099.2;
      O     ;
      A     M   7704.5;
      AN    I      0.1;
      AN    I     80.1;
      )     ;
      AN    M      3.3;
      =     M   7704.5;
      A     L      0.0;
      A(    ;
      A     I      7.1;
      A     DB327.DBX 1101.2;
      O     ;
      A     M   7704.6;
      AN    I      0.1;
      AN    I     80.1;
      )     ;
      AN    M      3.3;
      =     M   7704.6;
      A     L      0.0;
      A(    ;
      A     I      7.1;
      A     DB327.DBX 1103.2;
      O     ;
      A     M   7704.7;
      AN    I      0.1;
      AN    I     80.1;
      )     ;
      AN    M      3.3;
      =     M   7704.7;
NETWORK
TITLE =PROFINET MODULE ERROR(150~159)
